// TIA Portal project "BatchSimulation_S71500_multiple_throat" (V15)

(* hardware
DEVICE "S71500/ET200MP station_1"  S7-1500 station
   slot 0: "Rail_0"  Rack  6ES7 590-1***0-0AA0
   slot 1: "PLC_2_BatchController"  CPU 1512C-1 PN  6ES7 512-1CK01-0AB0  V2.5
      slot 3: "CPU display_1"  6ES7591-1AA00-0AA0
   slot 2: "CM PtP RS422/485 HF_1"  CM PtP RS422/485 HF  6ES7 541-1AB00-0AB0  V1.0
DEVICE "S71500/ET200MP station_2"  S7-1500 station
   slot 0: "Rail_0"  Rack  6ES7 590-1***0-0AA0
   slot 1: "PLC_1_Master"  CPU 1512C-1 PN  6ES7 512-1CK01-0AB0  V2.5
      slot 3: "CPU display_1"  6ES7591-1AA00-0AA0
*)

// ===== PLC "PLC_2_BatchController"  CPU 1512C-1 PN =====

VAR_GLOBAL   // PLC tag table "Default tag table"
   "System_Byte" AT %MB1 : Byte;
   "FirstScan" AT %M1.0 : Bool;
   "DiagStatusUpdate" AT %M1.1 : Bool;
   "AlwaysTRUE" AT %M1.2 : Bool;
   "AlwaysFALSE" AT %M1.3 : Bool;
END_VAR

DATA_BLOCK "Batch1_Send"   // DB4
{ S7_Optimized_Access := 'FALSE' }
VERSION : 0.1
   VAR
      Ready : Bool;   // Batch đã sẵn sàng
      Running : Bool;   // Batch đang chạy
      Clock : Bool;   // xung trả về từ cảm biến lưu lượng
      Pulse : Int := 13;   // tổng số xung từ lúc bắt đầu chạy của cảm biến lưu lượng
      Vout : Real;   // thể tích đã xuất ra (m3)
      ctrvalue : Real;   // độ mở van (0-100%)
   END_VAR
BEGIN
END_DATA_BLOCK

DATA_BLOCK "Batch1_Recv"   // DB5
{ S7_Optimized_Access := 'FALSE' }
VERSION : 0.1
   VAR
      Start : Bool;   // tín hiệu bắt đầu chạy
      Estop : Bool;   // tín hiệu dừng khẩn cấp
      Enable : Bool;   // tín hiệu cho phép làm việc
      PS : Int;   // số xung/lit của cảm biến lưu lượng
      Setpoint : Real;   // thể tích cần xuất
   END_VAR
BEGIN
END_DATA_BLOCK

DATA_BLOCK "Batch2_Send"   // DB8
{ S7_Optimized_Access := 'FALSE' }
VERSION : 0.1
   VAR
      Ready : Bool;   // Batch đã sẵn sàng
      Running : Bool;   // Batch đang chạy
      Clock : Bool;   // xung trả về từ cảm biến lưu lượng
      Pulse : Int := 13;   // tổng số xung từ lúc bắt đầu chạy của cảm biến lưu lượng
      Vout : Real;   // thể tích đã xuất ra (m3)
      ctrvalue : Real;   // độ mở van (0-100%)
   END_VAR
BEGIN
END_DATA_BLOCK

DATA_BLOCK "Batch2_Recv"   // DB9
{ S7_Optimized_Access := 'FALSE' }
VERSION : 0.1
   VAR
      Start : Bool;   // tín hiệu bắt đầu chạy
      Estop : Bool;   // tín hiệu dừng khẩn cấp
      Enable : Bool;   // tín hiệu cho phép làm việc
      PS : Int;   // số xung/lit của cảm biến lưu lượng
      Setpoint : Real;   // thể tích cần xuất
   END_VAR
BEGIN
END_DATA_BLOCK

DATA_BLOCK "RON921_Recv"   // DB12
{ S7_Optimized_Access := 'FALSE' }
VERSION : 0.1
   VAR
      Start : Bool;   // tín hiệu bắt đầu chạy
      Estop : Bool;   // tín hiệu dừng khẩn cấp
      Enable : Bool;   // tín hiệu cho phép làm việc
      PS : Int;   // số xung/lit của cảm biến lưu lượng
      Setpoint : Real;   // thể tích cần xuất
   END_VAR
BEGIN
END_DATA_BLOCK

DATA_BLOCK "RON921_Send"   // DB13
{ S7_Optimized_Access := 'FALSE' }
VERSION : 0.1
   VAR
      Ready : Bool;   // Batch đã sẵn sàng
      Running : Bool;   // Batch đang chạy
      Clock : Bool;   // xung trả về từ cảm biến lưu lượng
      Pulse : Int := 13;   // tổng số xung từ lúc bắt đầu chạy của cảm biến lưu lượng
      Vout : Real;   // thể tích đã xuất ra (m3)
      ctrvalue : Real;   // độ mở van (0-100%)
   END_VAR
BEGIN
END_DATA_BLOCK

DATA_BLOCK "RON922_Recv"   // DB14
{ S7_Optimized_Access := 'FALSE' }
VERSION : 0.1
   VAR
      Start : Bool;   // tín hiệu bắt đầu chạy
      Estop : Bool;   // tín hiệu dừng khẩn cấp
      Enable : Bool;   // tín hiệu cho phép làm việc
      PS : Int;   // số xung/lit của cảm biến lưu lượng
      Setpoint : Real;   // thể tích cần xuất
   END_VAR
BEGIN
END_DATA_BLOCK

DATA_BLOCK "RON922_Send"   // DB15
{ S7_Optimized_Access := 'FALSE' }
VERSION : 0.1
   VAR
      Ready : Bool;   // Batch đã sẵn sàng
      Running : Bool;   // Batch đang chạy
      Clock : Bool;   // xung trả về từ cảm biến lưu lượng
      Pulse : Int := 13;   // tổng số xung từ lúc bắt đầu chạy của cảm biến lưu lượng
      Vout : Real;   // thể tích đã xuất ra (m3)
      ctrvalue : Real;   // độ mở van (0-100%)
   END_VAR
BEGIN
END_DATA_BLOCK

DATA_BLOCK "RON951_Recv"   // DB20
{ S7_Optimized_Access := 'FALSE' }
VERSION : 0.1
   VAR
      Start : Bool;   // tín hiệu bắt đầu chạy
      Estop : Bool;   // tín hiệu dừng khẩn cấp
      Enable : Bool;   // tín hiệu cho phép làm việc
      PS : Int;   // số xung/lit của cảm biến lưu lượng
      Setpoint : Real;   // thể tích cần xuất
   END_VAR
BEGIN
END_DATA_BLOCK

DATA_BLOCK "RON951_Send"   // DB21
{ S7_Optimized_Access := 'FALSE' }
VERSION : 0.1
   VAR
      Ready : Bool;   // Batch đã sẵn sàng
      Running : Bool;   // Batch đang chạy
      Clock : Bool;   // xung trả về từ cảm biến lưu lượng
      Pulse : Int := 13;   // tổng số xung từ lúc bắt đầu chạy của cảm biến lưu lượng
      Vout : Real;   // thể tích đã xuất ra (m3)
      ctrvalue : Real;   // độ mở van (0-100%)
   END_VAR
BEGIN
END_DATA_BLOCK

DATA_BLOCK "RON952_Recv"   // DB22
{ S7_Optimized_Access := 'FALSE' }
VERSION : 0.1
   VAR
      Start : Bool;   // tín hiệu bắt đầu chạy
      Estop : Bool;   // tín hiệu dừng khẩn cấp
      Enable : Bool;   // tín hiệu cho phép làm việc
      PS : Int;   // số xung/lit của cảm biến lưu lượng
      Setpoint : Real;   // thể tích cần xuất
   END_VAR
BEGIN
END_DATA_BLOCK

DATA_BLOCK "RON952_Send"   // DB23
{ S7_Optimized_Access := 'FALSE' }
VERSION : 0.1
   VAR
      Ready : Bool;   // Batch đã sẵn sàng
      Running : Bool;   // Batch đang chạy
      Clock : Bool;   // xung trả về từ cảm biến lưu lượng
      Pulse : Int := 13;   // tổng số xung từ lúc bắt đầu chạy của cảm biến lưu lượng
      Vout : Real;   // thể tích đã xuất ra (m3)
      ctrvalue : Real;   // độ mở van (0-100%)
   END_VAR
BEGIN
END_DATA_BLOCK

DATA_BLOCK "E51_Recv"   // DB28
{ S7_Optimized_Access := 'FALSE' }
VERSION : 0.1
   VAR
      Start : Bool;   // tín hiệu bắt đầu chạy
      Estop : Bool;   // tín hiệu dừng khẩn cấp
      Enable : Bool;   // tín hiệu cho phép làm việc
      PS : Int := 13;   // số xung/lit của cảm biến lưu lượng
      Setpoint : Real;   // thể tích cần xuất
   END_VAR
BEGIN
END_DATA_BLOCK

DATA_BLOCK "E51_Send"   // DB29
{ S7_Optimized_Access := 'FALSE' }
VERSION : 0.1
   VAR
      Ready : Bool;   // Batch đã sẵn sàng
      Running : Bool;   // Batch đang chạy
      ClockRON92 : Bool;   // xung trả về từ cảm biến lưu lượng
      ClockE100 : Bool;
      PulseRON92 : Int := 13;   // tổng số xung từ lúc bắt đầu chạy của cảm biến lưu lượng
      PulseE100 : Int := 13;   // tổng số xung từ lúc bắt đầu chạy của cảm biến lưu lượng
      VoutRON92 : Real;   // thể tích đã xuất ra (m3)
      VoutE100 : Real;   // thể tích đã xuất ra (m3)
      Vout : Real;   // thể tích đã xuất ra (m3)
      ctrvalueRON92 : Real;   // độ mở van (0-100%)
      ctrvalueE100 : Real;   // độ mở van (0-100%)
   END_VAR
BEGIN
END_DATA_BLOCK

DATA_BLOCK "E52_Recv"   // DB30
{ S7_Optimized_Access := 'FALSE' }
VERSION : 0.1
   VAR
      Start : Bool;   // tín hiệu bắt đầu chạy
      Estop : Bool;   // tín hiệu dừng khẩn cấp
      Enable : Bool;   // tín hiệu cho phép làm việc
      PS : Int := 13;   // số xung/lit của cảm biến lưu lượng
      Setpoint : Real;   // thể tích cần xuất
   END_VAR
BEGIN
END_DATA_BLOCK

DATA_BLOCK "E52_Send"   // DB31
{ S7_Optimized_Access := 'FALSE' }
VERSION : 0.1
   VAR
      Ready : Bool;   // Batch đã sẵn sàng
      Running : Bool;   // Batch đang chạy
      ClockRON92 : Bool;   // xung trả về từ cảm biến lưu lượng
      ClockE100 : Bool;
      PulseRON92 : Int := 13;   // tổng số xung từ lúc bắt đầu chạy của cảm biến lưu lượng
      PulseE100 : Int := 13;   // tổng số xung từ lúc bắt đầu chạy của cảm biến lưu lượng
      VoutRON92 : Real;   // thể tích đã xuất ra (m3)
      VoutE100 : Real;   // thể tích đã xuất ra (m3)
      Vout : Real;   // thể tích đã xuất ra (m3)
      ctrvalueRON92 : Real;   // độ mở van (0-100%)
      ctrvalueE100 : Real;   // độ mở van (0-100%)
   END_VAR
BEGIN
END_DATA_BLOCK

// folder: System blocks/Program resources

DATA_BLOCK "IEC_Timer_0_DB"   // DB1
{ S7_Optimized_Access := 'TRUE' }
AUTHOR : Simatic
FAMILY : IEC
NAME : IEC_TMR
VERSION : 1.0
// stored: InstanceOfName IEC_TIMER
"IEC_TIMER"
BEGIN
END_DATA_BLOCK

DATA_BLOCK "IEC_Timer_0_DB_1"   // DB2
{ S7_Optimized_Access := 'TRUE' }
AUTHOR : Simatic
FAMILY : IEC
NAME : IEC_TMR
VERSION : 1.0
// stored: InstanceOfName IEC_TIMER
"IEC_TIMER"
BEGIN
END_DATA_BLOCK

// folder: (top level)

FUNCTION "ClockGenerator" : Void   // FC1, LAD
{ S7_Optimized_Access := 'TRUE' }
VERSION : 0.1
   VAR_INPUT
      "Flow (m3/h)" : Real;
      PS : Int;
   END_VAR
   VAR_IN_OUT
      clock : Bool;
   END_VAR
   VAR_TEMP
      timing_ms : Int;
      timing : Time;
   END_VAR
BEGIN

REGION Network 1: tính ra chu kì của xung theo lưu lượng
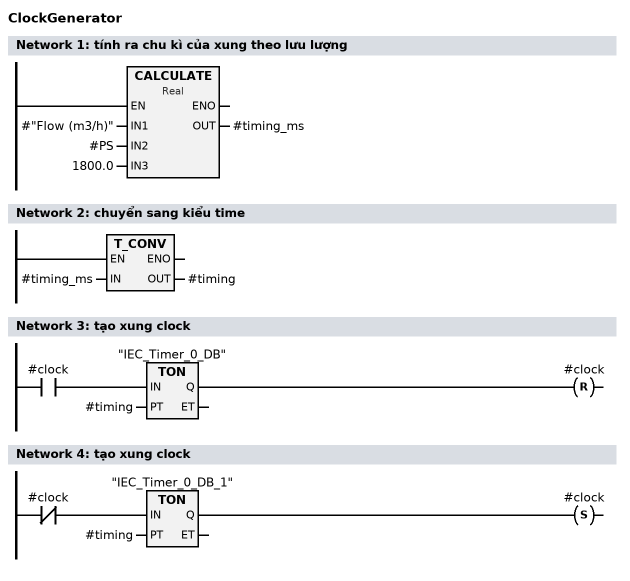
   RUNG wire#powerrail
      { S7_Templates := "SrcType := Real"; S7_Expression := "IN3/(IN1*IN2)" } Calculate(in1 := #"Flow (m3/h)", in2 := #PS, in3 := 1800.0, out => #timing_ms)
   END_RUNG
   // the same network as SCL:
   #timing_ms := 1800.0/(#"Flow (m3/h)"*#PS);
END_REGION

REGION Network 2: chuyển sang kiểu time
   #timing := T_CONV(IN := #timing_ms);
END_REGION

REGION Network 3: tạo xung clock
   "IEC_Timer_0_DB".TON(IN := #clock, PT := #timing);
   IF "IEC_Timer_0_DB".Q THEN #clock := FALSE; END_IF;
END_REGION

REGION Network 4: tạo xung clock
   "IEC_Timer_0_DB_1".TON(IN := NOT #clock, PT := #timing);
   IF "IEC_Timer_0_DB_1".Q THEN #clock := TRUE; END_IF;
END_REGION
END_FUNCTION

FUNCTION "BatchSimulation" : Void   // FC2, LAD
{ S7_Optimized_Access := 'TRUE' }
VERSION : 0.1
   VAR_INPUT
      Enable : Bool;
      Start : Bool;
      Estop : Bool;
      Setpoint : Real;
      PS : Int;
   END_VAR
   VAR_OUTPUT
      Ready : Bool;
   END_VAR
   VAR_IN_OUT
      "Vout(m3)" : Real;
      Running : Bool;
      pulse : Int;
      ctrlvalue : Real;
      clock : Bool;
   END_VAR
   VAR_TEMP
      flow : Real;
      tmp_clock : Bool;
      tmp_running : Bool;
   END_VAR
   VAR_TEMP   // added for the SCL form of the ladder/FBD networks
      _w1 : Bool;
   END_VAR
BEGIN

REGION Network 1: logic control
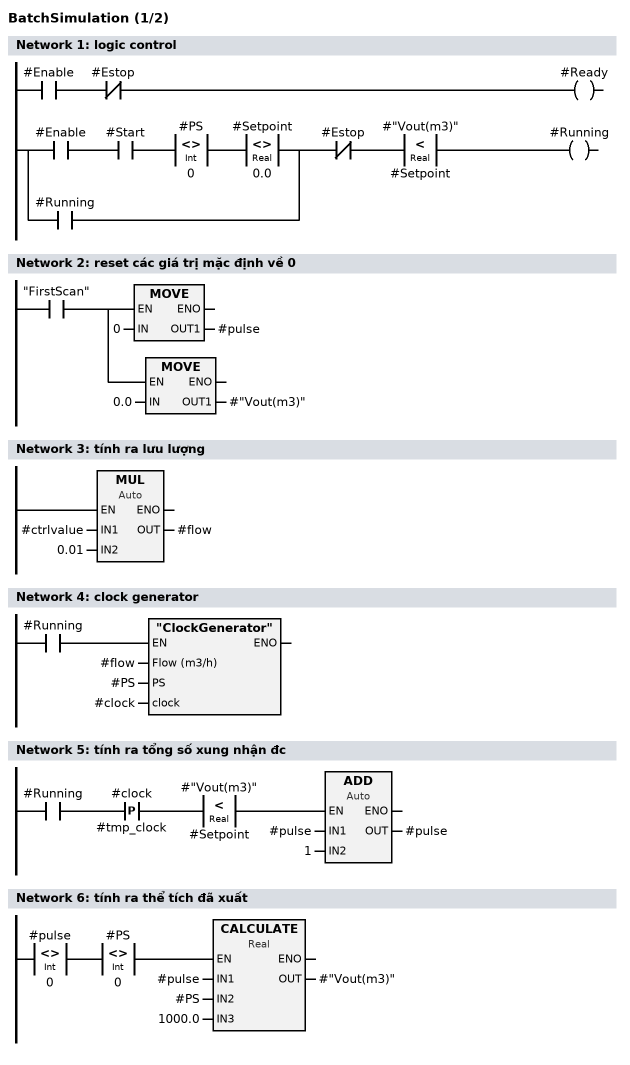
   RUNG wire#powerrail
      Contact( #Enable )
      I_Contact( #Estop )
      Coil( #Ready )
   END_RUNG
   RUNG wire#powerrail
      Contact( #Enable )
      Contact( #Start )
      { S7_Templates := "SrcType := Int" } NE_Contact(in1 := #PS, in2 := 0)
      { S7_Templates := "SrcType := Real" } NE_Contact(in1 := #Setpoint, in2 := 0.0)
      wire#w1
      I_Contact( #Estop )
      { S7_Templates := "SrcType := Real" } LT_Contact(in1 := #"Vout(m3)", in2 := #Setpoint)
      Coil( #Running )
   END_RUNG
   RUNG wire#powerrail
      Contact( #Running )
   END_RUNG wire#w1
   // the same network as SCL:
   #Ready := #Enable AND NOT #Estop;
   #Running := ((#Enable AND #Start AND (#PS <> 0) AND (#Setpoint <> 0.0)) OR #Running) AND NOT #Estop AND (#"Vout(m3)" < #Setpoint);
END_REGION

REGION Network 2: reset các giá trị mặc định về 0
   RUNG wire#powerrail
      Contact( "FirstScan" )
      wire#w1
      Move(in := 0, out1 => #pulse)
   END_RUNG
   RUNG wire#w1
      Move(in := 0.0, out1 => #"Vout(m3)")
   END_RUNG
   // the same network as SCL:
   IF "FirstScan" THEN
       #pulse := 0;
       #"Vout(m3)" := 0.0;
   END_IF;
END_REGION

REGION Network 3: tính ra lưu lượng
   RUNG wire#powerrail
      Mul(in1 := #ctrlvalue, in2 := 0.01, out => #flow)
   END_RUNG
   // the same network as SCL:
   #flow := #ctrlvalue * 0.01;
END_REGION

REGION Network 4: clock generator
   RUNG wire#powerrail
      Contact( #Running )
      "ClockGenerator"("Flow (m3/h)" := #flow, PS := #PS, clock := #clock)
   END_RUNG
   // the same network as SCL:
   IF #Running THEN "ClockGenerator"("Flow (m3/h)" := #flow, PS := #PS, clock := #clock); END_IF;
END_REGION

REGION Network 5: tính ra tổng số xung nhận đc
   RUNG wire#powerrail
      Contact( #Running )
      P_Contact(operand := #clock, bit := #tmp_clock)
      { S7_Templates := "SrcType := Real" } LT_Contact(in1 := #"Vout(m3)", in2 := #Setpoint)
      Add(in1 := #pulse, in2 := 1, out => #pulse)
   END_RUNG
   // the same network as SCL:
   #_w1 := #Running AND #clock AND NOT #tmp_clock;   // rising edge of #clock
   #tmp_clock := #clock;
   IF #_w1 AND (#"Vout(m3)" < #Setpoint) THEN #pulse := #pulse + 1; END_IF;
END_REGION

REGION Network 6: tính ra thể tích đã xuất
   RUNG wire#powerrail
      { S7_Templates := "SrcType := Int" } NE_Contact(in1 := #pulse, in2 := 0)
      { S7_Templates := "SrcType := Int" } NE_Contact(in1 := #PS, in2 := 0)
      { S7_Templates := "SrcType := Real"; S7_Expression := "(IN1/IN2)/IN3" } Calculate(in1 := #pulse, in2 := #PS, in3 := 1000.0, out => #"Vout(m3)")
   END_RUNG
   // the same network as SCL:
   IF (#pulse <> 0) AND (#PS <> 0) THEN #"Vout(m3)" := (#pulse/#PS)/1000.0; END_IF;
END_REGION

REGION Network 7: bộ PID điều khiển độ mở van
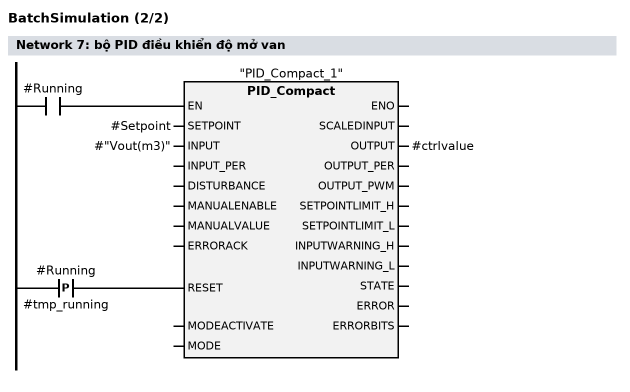
   #_w1 := #Running AND NOT #tmp_running;   // rising edge of #Running
   #tmp_running := #Running;
   IF #Running THEN
       "PID_Compact_1"(Setpoint := #Setpoint, Input := #"Vout(m3)", Reset := #_w1, Output => #ctrlvalue);   // PID_Compact
   END_IF;
END_REGION
END_FUNCTION

FUNCTION "DiezelProcess" : Void   // FC3, LAD
{ S7_Optimized_Access := 'TRUE' }
VERSION : 0.1
BEGIN

REGION Network 1: nhận dữ liệu từ DB của PLC họng 1
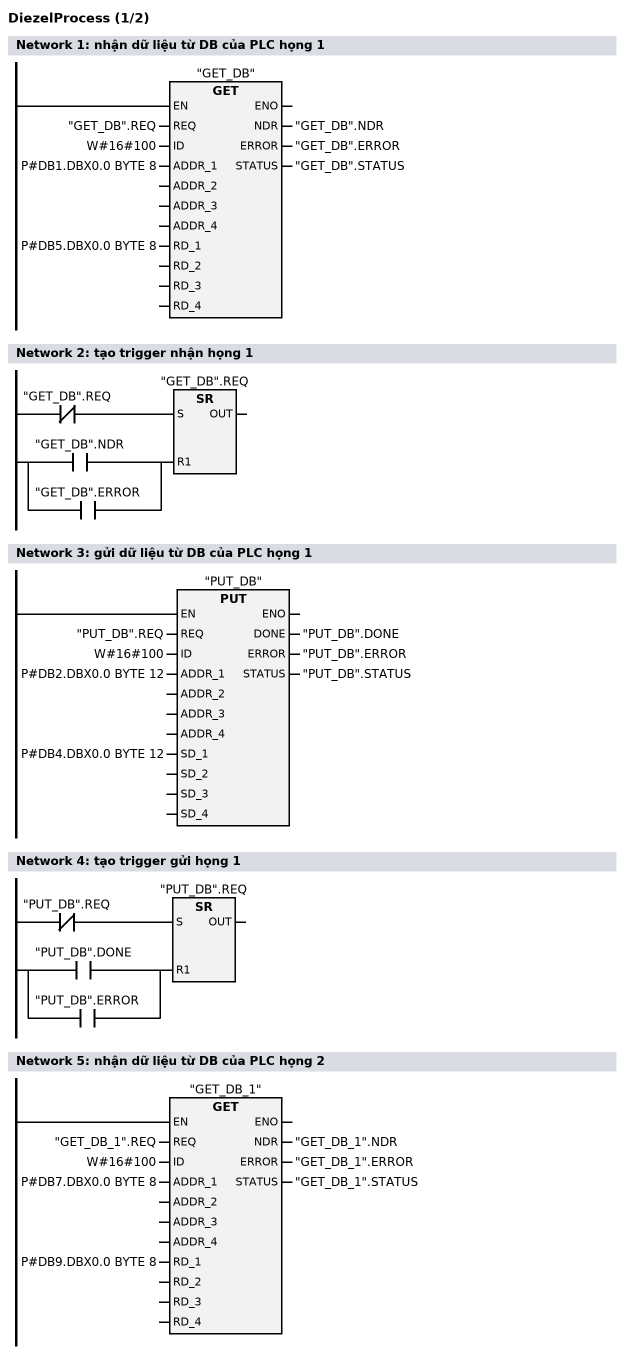
   "GET_DB"(REQ := "GET_DB".REQ,   // GET
            ID := W#16#100,
            ADDR_1 := P#DB1.DBX0.0 BYTE 8,
            RD_1 := P#DB5.DBX0.0 BYTE 8,
            NDR => "GET_DB".NDR,
            ERROR => "GET_DB".ERROR,
            STATUS => "GET_DB".STATUS);
END_REGION

REGION Network 2: tạo trigger nhận họng 1
   RUNG wire#powerrail
      I_Contact( "GET_DB".REQ )
      S_SR(operand := "GET_DB".REQ, r1 := wire#w1)
   END_RUNG
   RUNG wire#powerrail
      Contact( "GET_DB".NDR )
   END_RUNG wire#w1
   RUNG wire#powerrail
      Contact( "GET_DB".ERROR )
   END_RUNG wire#w1
   // the same network as SCL:
   IF NOT "GET_DB".REQ THEN
       "GET_DB".REQ := TRUE;   // SR flip-flop
   END_IF;
   IF "GET_DB".NDR OR "GET_DB".ERROR THEN "GET_DB".REQ := FALSE; END_IF;
END_REGION

REGION Network 3: gửi dữ liệu từ DB của PLC họng 1
   "PUT_DB"(REQ := "PUT_DB".REQ,   // PUT
            ID := W#16#100,
            ADDR_1 := P#DB2.DBX0.0 BYTE 12,
            SD_1 := P#DB4.DBX0.0 BYTE 12,
            DONE => "PUT_DB".DONE,
            ERROR => "PUT_DB".ERROR,
            STATUS => "PUT_DB".STATUS);
END_REGION

REGION Network 4: tạo trigger gửi họng 1
   RUNG wire#powerrail
      I_Contact( "PUT_DB".REQ )
      S_SR(operand := "PUT_DB".REQ, r1 := wire#w1)
   END_RUNG
   RUNG wire#powerrail
      Contact( "PUT_DB".DONE )
   END_RUNG wire#w1
   RUNG wire#powerrail
      Contact( "PUT_DB".ERROR )
   END_RUNG wire#w1
   // the same network as SCL:
   IF NOT "PUT_DB".REQ THEN
       "PUT_DB".REQ := TRUE;   // SR flip-flop
   END_IF;
   IF "PUT_DB".DONE OR "PUT_DB".ERROR THEN "PUT_DB".REQ := FALSE; END_IF;
END_REGION

REGION Network 5: nhận dữ liệu từ DB của PLC họng 2
   "GET_DB_1"(REQ := "GET_DB_1".REQ,   // GET
              ID := W#16#100,
              ADDR_1 := P#DB7.DBX0.0 BYTE 8,
              RD_1 := P#DB9.DBX0.0 BYTE 8,
              NDR => "GET_DB_1".NDR,
              ERROR => "GET_DB_1".ERROR,
              STATUS => "GET_DB_1".STATUS);
END_REGION

REGION Network 6: tạo trigger nhận họng 2
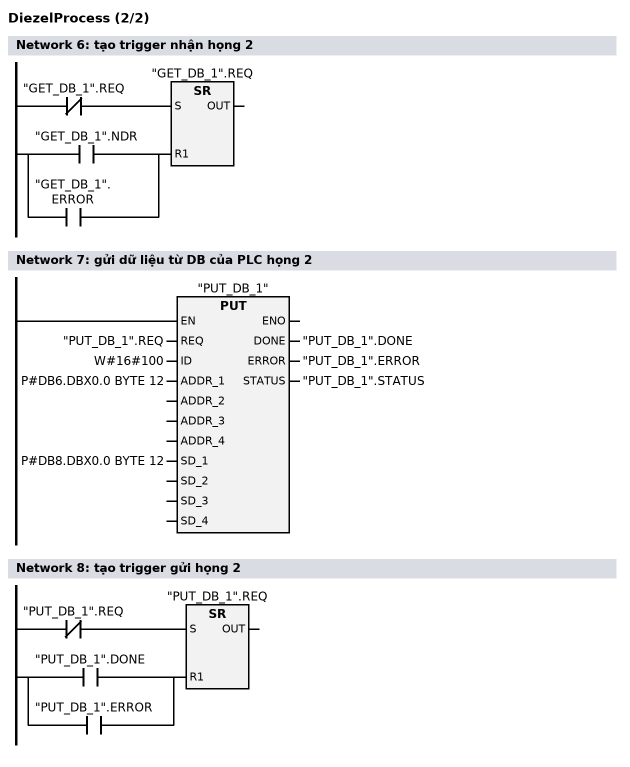
   RUNG wire#powerrail
      I_Contact( "GET_DB_1".REQ )
      S_SR(operand := "GET_DB_1".REQ, r1 := wire#w1)
   END_RUNG
   RUNG wire#powerrail
      Contact( "GET_DB_1".NDR )
   END_RUNG wire#w1
   RUNG wire#powerrail
      Contact( "GET_DB_1".ERROR )
   END_RUNG wire#w1
   // the same network as SCL:
   IF NOT "GET_DB_1".REQ THEN
       "GET_DB_1".REQ := TRUE;   // SR flip-flop
   END_IF;
   IF "GET_DB_1".NDR OR "GET_DB_1".ERROR THEN "GET_DB_1".REQ := FALSE; END_IF;
END_REGION

REGION Network 7: gửi dữ liệu từ DB của PLC họng 2
   "PUT_DB_1"(REQ := "PUT_DB_1".REQ,   // PUT
              ID := W#16#100,
              ADDR_1 := P#DB6.DBX0.0 BYTE 12,
              SD_1 := P#DB8.DBX0.0 BYTE 12,
              DONE => "PUT_DB_1".DONE,
              ERROR => "PUT_DB_1".ERROR,
              STATUS => "PUT_DB_1".STATUS);
END_REGION

REGION Network 8: tạo trigger gửi họng 2
   RUNG wire#powerrail
      I_Contact( "PUT_DB_1".REQ )
      S_SR(operand := "PUT_DB_1".REQ, r1 := wire#w1)
   END_RUNG
   RUNG wire#powerrail
      Contact( "PUT_DB_1".DONE )
   END_RUNG wire#w1
   RUNG wire#powerrail
      Contact( "PUT_DB_1".ERROR )
   END_RUNG wire#w1
   // the same network as SCL:
   IF NOT "PUT_DB_1".REQ THEN
       "PUT_DB_1".REQ := TRUE;   // SR flip-flop
   END_IF;
   IF "PUT_DB_1".DONE OR "PUT_DB_1".ERROR THEN "PUT_DB_1".REQ := FALSE; END_IF;
END_REGION
END_FUNCTION

FUNCTION "RON92Process" : Void   // FC4, LAD
{ S7_Optimized_Access := 'TRUE' }
VERSION : 0.1
BEGIN

REGION Network 1: nhận dữ liệu từ DB của PLC họng 1
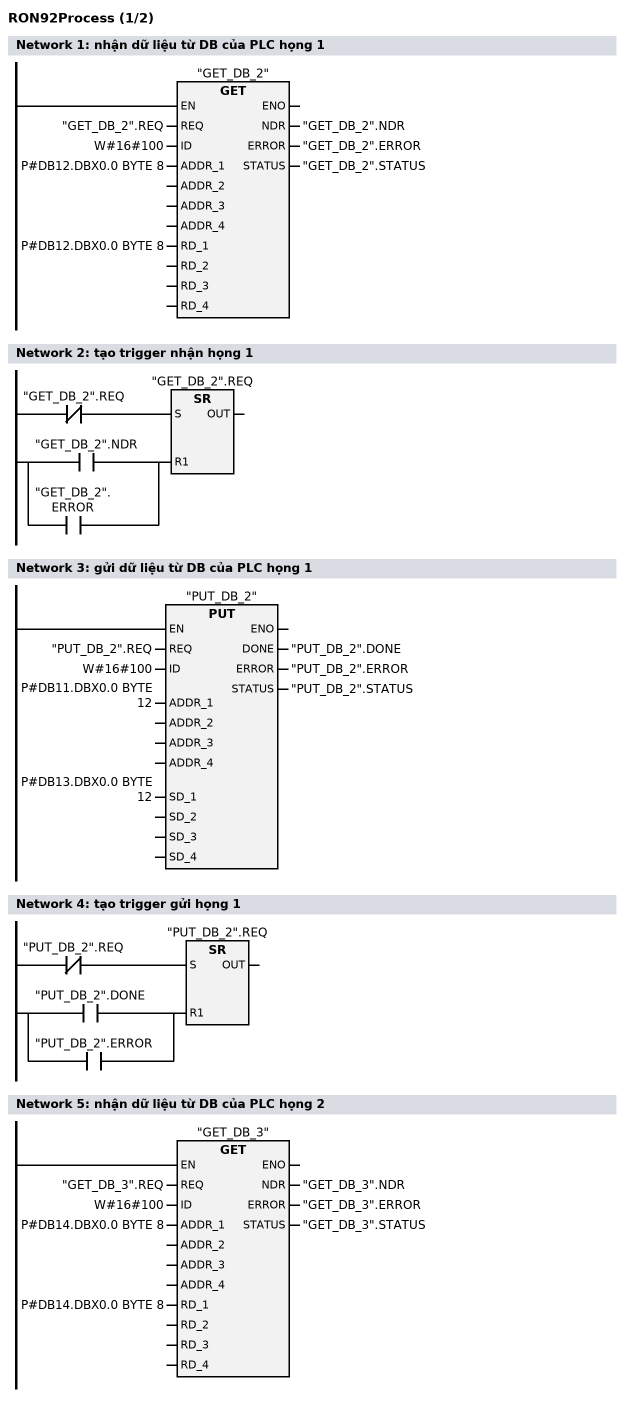
   "GET_DB_2"(REQ := "GET_DB_2".REQ,   // GET
              ID := W#16#100,
              ADDR_1 := P#DB12.DBX0.0 BYTE 8,
              RD_1 := P#DB12.DBX0.0 BYTE 8,
              NDR => "GET_DB_2".NDR,
              ERROR => "GET_DB_2".ERROR,
              STATUS => "GET_DB_2".STATUS);
END_REGION

REGION Network 2: tạo trigger nhận họng 1
   RUNG wire#powerrail
      I_Contact( "GET_DB_2".REQ )
      S_SR(operand := "GET_DB_2".REQ, r1 := wire#w1)
   END_RUNG
   RUNG wire#powerrail
      Contact( "GET_DB_2".NDR )
   END_RUNG wire#w1
   RUNG wire#powerrail
      Contact( "GET_DB_2".ERROR )
   END_RUNG wire#w1
   // the same network as SCL:
   IF NOT "GET_DB_2".REQ THEN
       "GET_DB_2".REQ := TRUE;   // SR flip-flop
   END_IF;
   IF "GET_DB_2".NDR OR "GET_DB_2".ERROR THEN "GET_DB_2".REQ := FALSE; END_IF;
END_REGION

REGION Network 3: gửi dữ liệu từ DB của PLC họng 1
   "PUT_DB_2"(REQ := "PUT_DB_2".REQ,   // PUT
              ID := W#16#100,
              ADDR_1 := P#DB11.DBX0.0 BYTE 12,
              SD_1 := P#DB13.DBX0.0 BYTE 12,
              DONE => "PUT_DB_2".DONE,
              ERROR => "PUT_DB_2".ERROR,
              STATUS => "PUT_DB_2".STATUS);
END_REGION

REGION Network 4: tạo trigger gửi họng 1
   RUNG wire#powerrail
      I_Contact( "PUT_DB_2".REQ )
      S_SR(operand := "PUT_DB_2".REQ, r1 := wire#w1)
   END_RUNG
   RUNG wire#powerrail
      Contact( "PUT_DB_2".DONE )
   END_RUNG wire#w1
   RUNG wire#powerrail
      Contact( "PUT_DB_2".ERROR )
   END_RUNG wire#w1
   // the same network as SCL:
   IF NOT "PUT_DB_2".REQ THEN
       "PUT_DB_2".REQ := TRUE;   // SR flip-flop
   END_IF;
   IF "PUT_DB_2".DONE OR "PUT_DB_2".ERROR THEN "PUT_DB_2".REQ := FALSE; END_IF;
END_REGION

REGION Network 5: nhận dữ liệu từ DB của PLC họng 2
   "GET_DB_3"(REQ := "GET_DB_3".REQ,   // GET
              ID := W#16#100,
              ADDR_1 := P#DB14.DBX0.0 BYTE 8,
              RD_1 := P#DB14.DBX0.0 BYTE 8,
              NDR => "GET_DB_3".NDR,
              ERROR => "GET_DB_3".ERROR,
              STATUS => "GET_DB_3".STATUS);
END_REGION

REGION Network 6: tạo trigger nhận họng 2
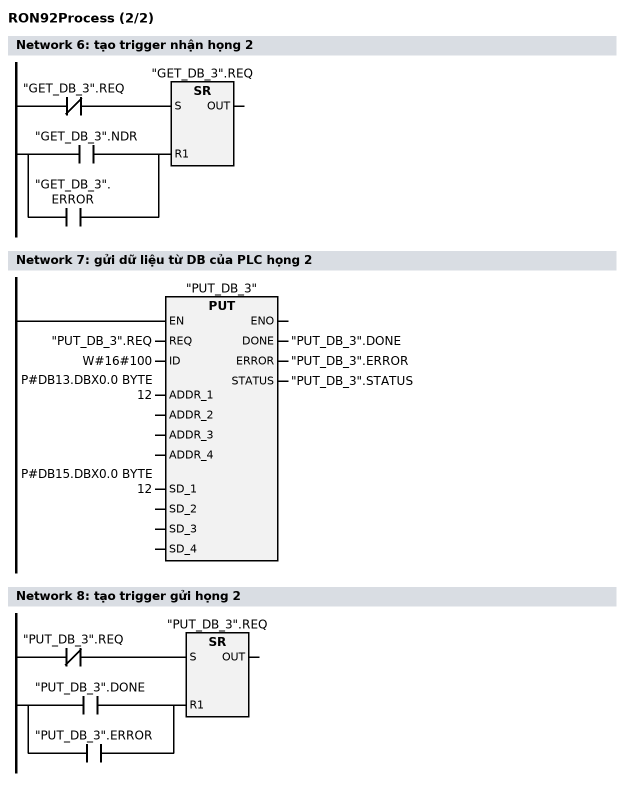
   RUNG wire#powerrail
      I_Contact( "GET_DB_3".REQ )
      S_SR(operand := "GET_DB_3".REQ, r1 := wire#w1)
   END_RUNG
   RUNG wire#powerrail
      Contact( "GET_DB_3".NDR )
   END_RUNG wire#w1
   RUNG wire#powerrail
      Contact( "GET_DB_3".ERROR )
   END_RUNG wire#w1
   // the same network as SCL:
   IF NOT "GET_DB_3".REQ THEN
       "GET_DB_3".REQ := TRUE;   // SR flip-flop
   END_IF;
   IF "GET_DB_3".NDR OR "GET_DB_3".ERROR THEN "GET_DB_3".REQ := FALSE; END_IF;
END_REGION

REGION Network 7: gửi dữ liệu từ DB của PLC họng 2
   "PUT_DB_3"(REQ := "PUT_DB_3".REQ,   // PUT
              ID := W#16#100,
              ADDR_1 := P#DB13.DBX0.0 BYTE 12,
              SD_1 := P#DB15.DBX0.0 BYTE 12,
              DONE => "PUT_DB_3".DONE,
              ERROR => "PUT_DB_3".ERROR,
              STATUS => "PUT_DB_3".STATUS);
END_REGION

REGION Network 8: tạo trigger gửi họng 2
   RUNG wire#powerrail
      I_Contact( "PUT_DB_3".REQ )
      S_SR(operand := "PUT_DB_3".REQ, r1 := wire#w1)
   END_RUNG
   RUNG wire#powerrail
      Contact( "PUT_DB_3".DONE )
   END_RUNG wire#w1
   RUNG wire#powerrail
      Contact( "PUT_DB_3".ERROR )
   END_RUNG wire#w1
   // the same network as SCL:
   IF NOT "PUT_DB_3".REQ THEN
       "PUT_DB_3".REQ := TRUE;   // SR flip-flop
   END_IF;
   IF "PUT_DB_3".DONE OR "PUT_DB_3".ERROR THEN "PUT_DB_3".REQ := FALSE; END_IF;
END_REGION
END_FUNCTION

FUNCTION "RON95Process" : Void   // FC5, LAD
{ S7_Optimized_Access := 'TRUE' }
VERSION : 0.1
BEGIN

REGION Network 1: nhận dữ liệu từ DB của PLC họng 1
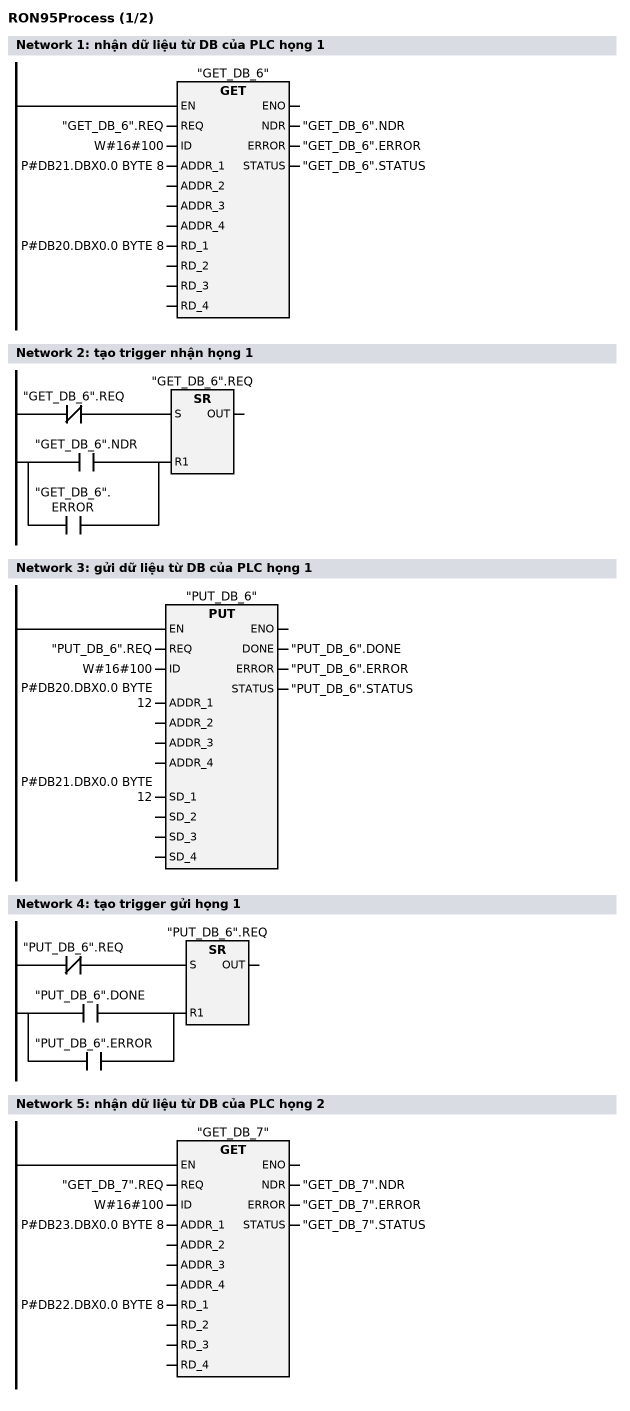
   "GET_DB_6"(REQ := "GET_DB_6".REQ,   // GET
              ID := W#16#100,
              ADDR_1 := P#DB21.DBX0.0 BYTE 8,
              RD_1 := P#DB20.DBX0.0 BYTE 8,
              NDR => "GET_DB_6".NDR,
              ERROR => "GET_DB_6".ERROR,
              STATUS => "GET_DB_6".STATUS);
END_REGION

REGION Network 2: tạo trigger nhận họng 1
   RUNG wire#powerrail
      I_Contact( "GET_DB_6".REQ )
      S_SR(operand := "GET_DB_6".REQ, r1 := wire#w1)
   END_RUNG
   RUNG wire#powerrail
      Contact( "GET_DB_6".NDR )
   END_RUNG wire#w1
   RUNG wire#powerrail
      Contact( "GET_DB_6".ERROR )
   END_RUNG wire#w1
   // the same network as SCL:
   IF NOT "GET_DB_6".REQ THEN
       "GET_DB_6".REQ := TRUE;   // SR flip-flop
   END_IF;
   IF "GET_DB_6".NDR OR "GET_DB_6".ERROR THEN "GET_DB_6".REQ := FALSE; END_IF;
END_REGION

REGION Network 3: gửi dữ liệu từ DB của PLC họng 1
   "PUT_DB_6"(REQ := "PUT_DB_6".REQ,   // PUT
              ID := W#16#100,
              ADDR_1 := P#DB20.DBX0.0 BYTE 12,
              SD_1 := P#DB21.DBX0.0 BYTE 12,
              DONE => "PUT_DB_6".DONE,
              ERROR => "PUT_DB_6".ERROR,
              STATUS => "PUT_DB_6".STATUS);
END_REGION

REGION Network 4: tạo trigger gửi họng 1
   RUNG wire#powerrail
      I_Contact( "PUT_DB_6".REQ )
      S_SR(operand := "PUT_DB_6".REQ, r1 := wire#w1)
   END_RUNG
   RUNG wire#powerrail
      Contact( "PUT_DB_6".DONE )
   END_RUNG wire#w1
   RUNG wire#powerrail
      Contact( "PUT_DB_6".ERROR )
   END_RUNG wire#w1
   // the same network as SCL:
   IF NOT "PUT_DB_6".REQ THEN
       "PUT_DB_6".REQ := TRUE;   // SR flip-flop
   END_IF;
   IF "PUT_DB_6".DONE OR "PUT_DB_6".ERROR THEN "PUT_DB_6".REQ := FALSE; END_IF;
END_REGION

REGION Network 5: nhận dữ liệu từ DB của PLC họng 2
   "GET_DB_7"(REQ := "GET_DB_7".REQ,   // GET
              ID := W#16#100,
              ADDR_1 := P#DB23.DBX0.0 BYTE 8,
              RD_1 := P#DB22.DBX0.0 BYTE 8,
              NDR => "GET_DB_7".NDR,
              ERROR => "GET_DB_7".ERROR,
              STATUS => "GET_DB_7".STATUS);
END_REGION

REGION Network 6: tạo trigger nhận họng 2
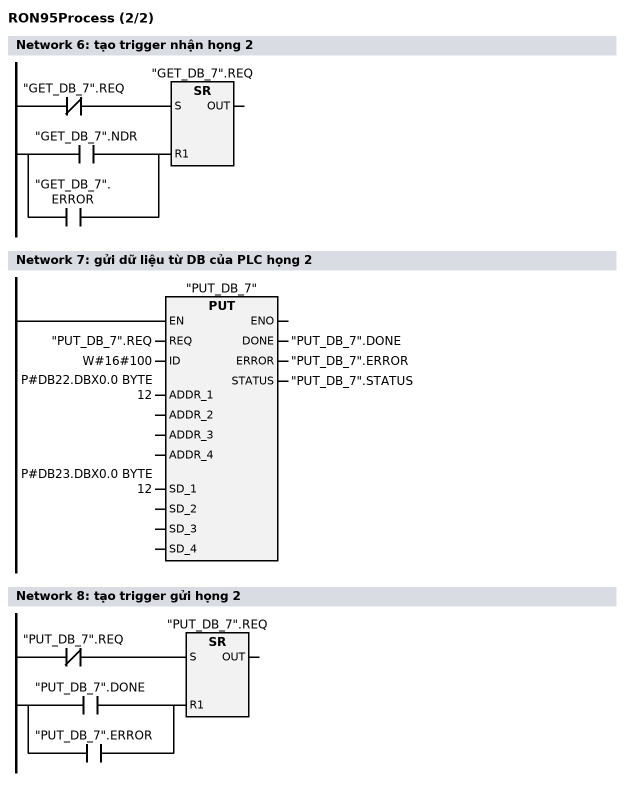
   RUNG wire#powerrail
      I_Contact( "GET_DB_7".REQ )
      S_SR(operand := "GET_DB_7".REQ, r1 := wire#w1)
   END_RUNG
   RUNG wire#powerrail
      Contact( "GET_DB_7".NDR )
   END_RUNG wire#w1
   RUNG wire#powerrail
      Contact( "GET_DB_7".ERROR )
   END_RUNG wire#w1
   // the same network as SCL:
   IF NOT "GET_DB_7".REQ THEN
       "GET_DB_7".REQ := TRUE;   // SR flip-flop
   END_IF;
   IF "GET_DB_7".NDR OR "GET_DB_7".ERROR THEN "GET_DB_7".REQ := FALSE; END_IF;
END_REGION

REGION Network 7: gửi dữ liệu từ DB của PLC họng 2
   "PUT_DB_7"(REQ := "PUT_DB_7".REQ,   // PUT
              ID := W#16#100,
              ADDR_1 := P#DB22.DBX0.0 BYTE 12,
              SD_1 := P#DB23.DBX0.0 BYTE 12,
              DONE => "PUT_DB_7".DONE,
              ERROR => "PUT_DB_7".ERROR,
              STATUS => "PUT_DB_7".STATUS);
END_REGION

REGION Network 8: tạo trigger gửi họng 2
   RUNG wire#powerrail
      I_Contact( "PUT_DB_7".REQ )
      S_SR(operand := "PUT_DB_7".REQ, r1 := wire#w1)
   END_RUNG
   RUNG wire#powerrail
      Contact( "PUT_DB_7".DONE )
   END_RUNG wire#w1
   RUNG wire#powerrail
      Contact( "PUT_DB_7".ERROR )
   END_RUNG wire#w1
   // the same network as SCL:
   IF NOT "PUT_DB_7".REQ THEN
       "PUT_DB_7".REQ := TRUE;   // SR flip-flop
   END_IF;
   IF "PUT_DB_7".DONE OR "PUT_DB_7".ERROR THEN "PUT_DB_7".REQ := FALSE; END_IF;
END_REGION
END_FUNCTION

FUNCTION "BatchSimulationE5" : Void   // FC6, LAD
{ S7_Optimized_Access := 'TRUE' }
VERSION : 0.1
   VAR_INPUT
      Enable : Bool;
      Start : Bool;
      Estop : Bool;
      Setpoint : Real;
      PS : Int;
   END_VAR
   VAR_OUTPUT
      Ready : Bool;
   END_VAR
   VAR_IN_OUT
      "Vout(m3)" : Real;
      "VoutRON92(m3)" : Real;
      "VoutE100(m3)" : Real;
      Running : Bool;
      pulseRON92 : Int;
      pulseE100 : Int;
      ctrlvalueRON92 : Real;
      ctrlvalueE100 : Real;
      clockRON92 : Bool;
      clockE100 : Bool;
   END_VAR
   VAR_TEMP
      flowRON92 : Real;
      flowE100 : Real;
      tmp_clock : Bool;
      tmp_running : Bool;
   END_VAR
   VAR_TEMP   // added for the SCL form of the ladder/FBD networks
      _w1 : Bool;
   END_VAR
BEGIN

REGION Network 1: logic control
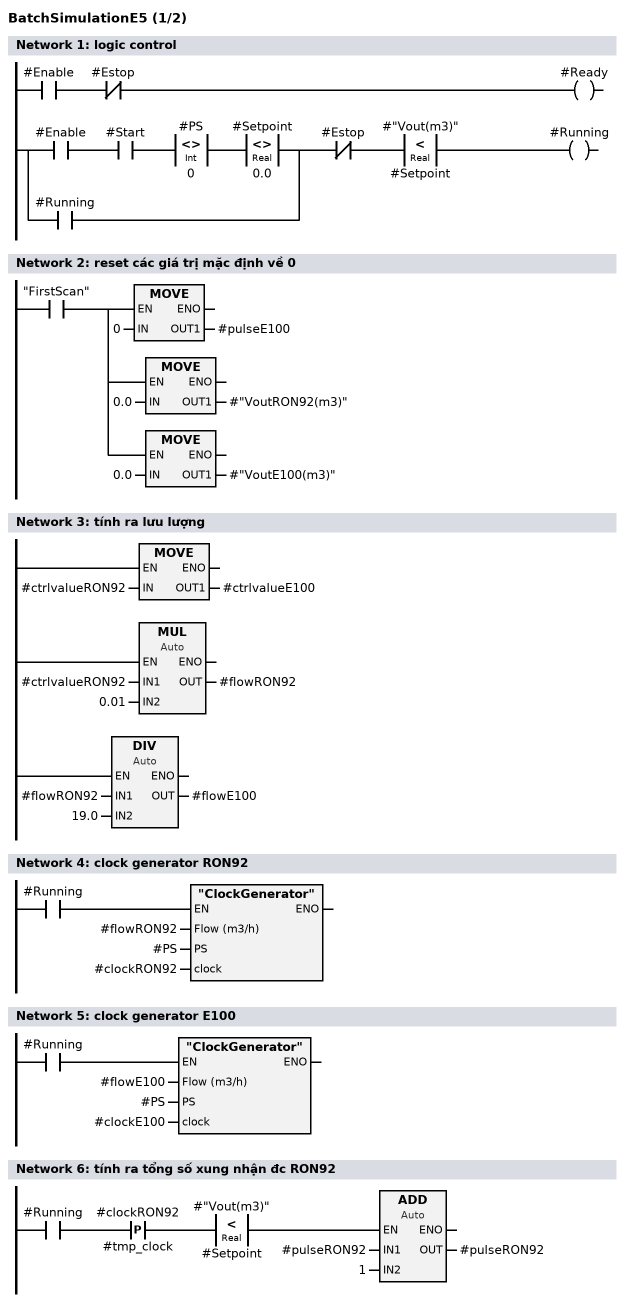
   RUNG wire#powerrail
      Contact( #Enable )
      I_Contact( #Estop )
      Coil( #Ready )
   END_RUNG
   RUNG wire#powerrail
      Contact( #Enable )
      Contact( #Start )
      { S7_Templates := "SrcType := Int" } NE_Contact(in1 := #PS, in2 := 0)
      { S7_Templates := "SrcType := Real" } NE_Contact(in1 := #Setpoint, in2 := 0.0)
      wire#w1
      I_Contact( #Estop )
      { S7_Templates := "SrcType := Real" } LT_Contact(in1 := #"Vout(m3)", in2 := #Setpoint)
      Coil( #Running )
   END_RUNG
   RUNG wire#powerrail
      Contact( #Running )
   END_RUNG wire#w1
   // the same network as SCL:
   #Ready := #Enable AND NOT #Estop;
   #Running := ((#Enable AND #Start AND (#PS <> 0) AND (#Setpoint <> 0.0)) OR #Running) AND NOT #Estop AND (#"Vout(m3)" < #Setpoint);
END_REGION

REGION Network 2: reset các giá trị mặc định về 0
   RUNG wire#powerrail
      Contact( "FirstScan" )
      wire#w1
      Move(in := 0, out1 => #pulseE100)
   END_RUNG
   RUNG wire#w1
      Move(in := 0.0, out1 => #"VoutRON92(m3)")
   END_RUNG
   RUNG wire#w1
      Move(in := 0.0, out1 => #"VoutE100(m3)")
   END_RUNG
   // the same network as SCL:
   IF "FirstScan" THEN
       #pulseE100 := 0;
       #"VoutRON92(m3)" := 0.0;
       #"VoutE100(m3)" := 0.0;
   END_IF;
END_REGION

REGION Network 3: tính ra lưu lượng
   RUNG wire#powerrail
      Move(in := #ctrlvalueRON92, out1 => #ctrlvalueE100)
   END_RUNG
   RUNG wire#powerrail
      Mul(in1 := #ctrlvalueRON92, in2 := 0.01, out => #flowRON92)
   END_RUNG
   RUNG wire#powerrail
      Div(in1 := #flowRON92, in2 := 19.0, out => #flowE100)
   END_RUNG
   // the same network as SCL:
   #ctrlvalueE100 := #ctrlvalueRON92;
   #flowRON92 := #ctrlvalueRON92 * 0.01;
   #flowE100 := #flowRON92 / 19.0;
END_REGION

REGION Network 4: clock generator RON92
   RUNG wire#powerrail
      Contact( #Running )
      "ClockGenerator"("Flow (m3/h)" := #flowRON92, PS := #PS, clock := #clockRON92)
   END_RUNG
   // the same network as SCL:
   IF #Running THEN "ClockGenerator"("Flow (m3/h)" := #flowRON92, PS := #PS, clock := #clockRON92); END_IF;
END_REGION

REGION Network 5: clock generator E100
   RUNG wire#powerrail
      Contact( #Running )
      "ClockGenerator"("Flow (m3/h)" := #flowE100, PS := #PS, clock := #clockE100)
   END_RUNG
   // the same network as SCL:
   IF #Running THEN "ClockGenerator"("Flow (m3/h)" := #flowE100, PS := #PS, clock := #clockE100); END_IF;
END_REGION

REGION Network 6: tính ra tổng số xung nhận đc RON92
   RUNG wire#powerrail
      Contact( #Running )
      P_Contact(operand := #clockRON92, bit := #tmp_clock)
      { S7_Templates := "SrcType := Real" } LT_Contact(in1 := #"Vout(m3)", in2 := #Setpoint)
      Add(in1 := #pulseRON92, in2 := 1, out => #pulseRON92)
   END_RUNG
   // the same network as SCL:
   #_w1 := #Running AND #clockRON92 AND NOT #tmp_clock;   // rising edge of #clockRON92
   #tmp_clock := #clockRON92;
   IF #_w1 AND (#"Vout(m3)" < #Setpoint) THEN #pulseRON92 := #pulseRON92 + 1; END_IF;
END_REGION

REGION Network 7: tính ra tổng số xung nhận đc E100
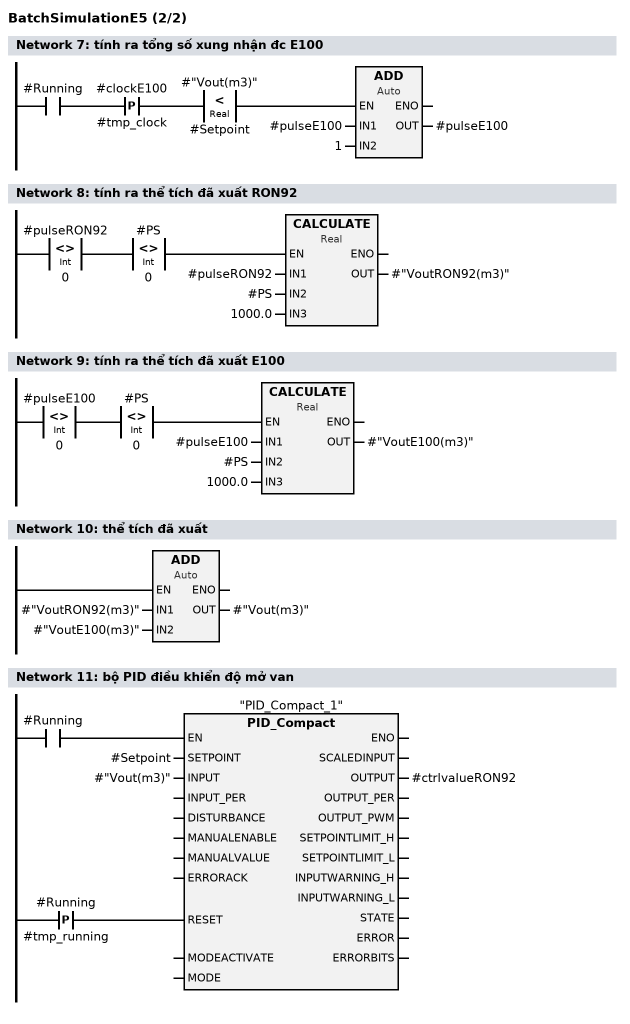
   RUNG wire#powerrail
      Contact( #Running )
      P_Contact(operand := #clockE100, bit := #tmp_clock)
      { S7_Templates := "SrcType := Real" } LT_Contact(in1 := #"Vout(m3)", in2 := #Setpoint)
      Add(in1 := #pulseE100, in2 := 1, out => #pulseE100)
   END_RUNG
   // the same network as SCL:
   #_w1 := #Running AND #clockE100 AND NOT #tmp_clock;   // rising edge of #clockE100
   #tmp_clock := #clockE100;
   IF #_w1 AND (#"Vout(m3)" < #Setpoint) THEN #pulseE100 := #pulseE100 + 1; END_IF;
END_REGION

REGION Network 8: tính ra thể tích đã xuất RON92
   RUNG wire#powerrail
      { S7_Templates := "SrcType := Int" } NE_Contact(in1 := #pulseRON92, in2 := 0)
      { S7_Templates := "SrcType := Int" } NE_Contact(in1 := #PS, in2 := 0)
      { S7_Templates := "SrcType := Real"; S7_Expression := "(IN1/IN2)/IN3" } Calculate(in1 := #pulseRON92, in2 := #PS, in3 := 1000.0, out => #"VoutRON92(m3)")
   END_RUNG
   // the same network as SCL:
   IF (#pulseRON92 <> 0) AND (#PS <> 0) THEN #"VoutRON92(m3)" := (#pulseRON92/#PS)/1000.0; END_IF;
END_REGION

REGION Network 9: tính ra thể tích đã xuất E100
   RUNG wire#powerrail
      { S7_Templates := "SrcType := Int" } NE_Contact(in1 := #pulseE100, in2 := 0)
      { S7_Templates := "SrcType := Int" } NE_Contact(in1 := #PS, in2 := 0)
      { S7_Templates := "SrcType := Real"; S7_Expression := "(IN1/IN2)/IN3" } Calculate(in1 := #pulseE100, in2 := #PS, in3 := 1000.0, out => #"VoutE100(m3)")
   END_RUNG
   // the same network as SCL:
   IF (#pulseE100 <> 0) AND (#PS <> 0) THEN #"VoutE100(m3)" := (#pulseE100/#PS)/1000.0; END_IF;
END_REGION

REGION Network 10: thể tích đã xuất
   RUNG wire#powerrail
      Add(in1 := #"VoutRON92(m3)", in2 := #"VoutE100(m3)", out => #"Vout(m3)")
   END_RUNG
   // the same network as SCL:
   #"Vout(m3)" := #"VoutRON92(m3)" + #"VoutE100(m3)";
END_REGION

REGION Network 11: bộ PID điều khiển độ mở van
   #_w1 := #Running AND NOT #tmp_running;   // rising edge of #Running
   #tmp_running := #Running;
   IF #Running THEN
       "PID_Compact_1"(Setpoint := #Setpoint, Input := #"Vout(m3)", Reset := #_w1, Output => #ctrlvalueRON92);   // PID_Compact
   END_IF;
END_REGION
END_FUNCTION

FUNCTION "E5Process" : Void   // FC7, LAD
{ S7_Optimized_Access := 'TRUE' }
VERSION : 0.1
BEGIN

REGION Network 1: nhận dữ liệu từ DB của PLC họng 1
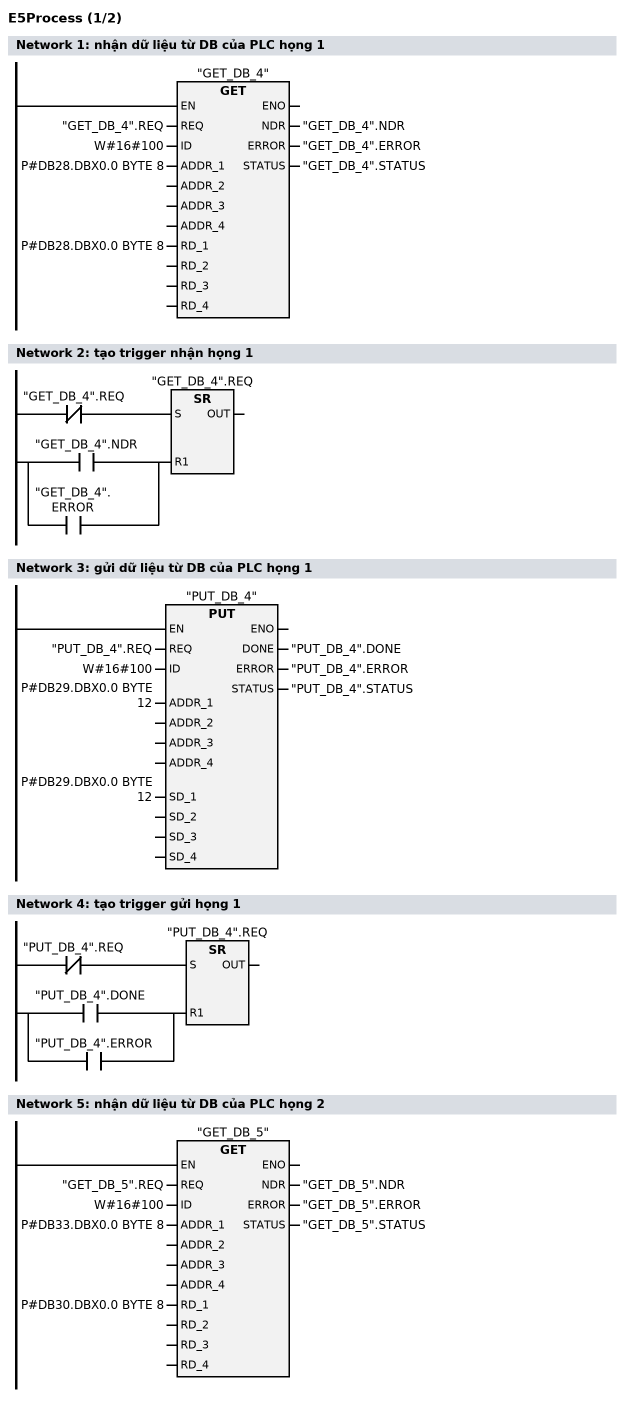
   "GET_DB_4"(REQ := "GET_DB_4".REQ,   // GET
              ID := W#16#100,
              ADDR_1 := P#DB28.DBX0.0 BYTE 8,
              RD_1 := P#DB28.DBX0.0 BYTE 8,
              NDR => "GET_DB_4".NDR,
              ERROR => "GET_DB_4".ERROR,
              STATUS => "GET_DB_4".STATUS);
END_REGION

REGION Network 2: tạo trigger nhận họng 1
   RUNG wire#powerrail
      I_Contact( "GET_DB_4".REQ )
      S_SR(operand := "GET_DB_4".REQ, r1 := wire#w1)
   END_RUNG
   RUNG wire#powerrail
      Contact( "GET_DB_4".NDR )
   END_RUNG wire#w1
   RUNG wire#powerrail
      Contact( "GET_DB_4".ERROR )
   END_RUNG wire#w1
   // the same network as SCL:
   IF NOT "GET_DB_4".REQ THEN
       "GET_DB_4".REQ := TRUE;   // SR flip-flop
   END_IF;
   IF "GET_DB_4".NDR OR "GET_DB_4".ERROR THEN "GET_DB_4".REQ := FALSE; END_IF;
END_REGION

REGION Network 3: gửi dữ liệu từ DB của PLC họng 1
   "PUT_DB_4"(REQ := "PUT_DB_4".REQ,   // PUT
              ID := W#16#100,
              ADDR_1 := P#DB29.DBX0.0 BYTE 12,
              SD_1 := P#DB29.DBX0.0 BYTE 12,
              DONE => "PUT_DB_4".DONE,
              ERROR => "PUT_DB_4".ERROR,
              STATUS => "PUT_DB_4".STATUS);
END_REGION

REGION Network 4: tạo trigger gửi họng 1
   RUNG wire#powerrail
      I_Contact( "PUT_DB_4".REQ )
      S_SR(operand := "PUT_DB_4".REQ, r1 := wire#w1)
   END_RUNG
   RUNG wire#powerrail
      Contact( "PUT_DB_4".DONE )
   END_RUNG wire#w1
   RUNG wire#powerrail
      Contact( "PUT_DB_4".ERROR )
   END_RUNG wire#w1
   // the same network as SCL:
   IF NOT "PUT_DB_4".REQ THEN
       "PUT_DB_4".REQ := TRUE;   // SR flip-flop
   END_IF;
   IF "PUT_DB_4".DONE OR "PUT_DB_4".ERROR THEN "PUT_DB_4".REQ := FALSE; END_IF;
END_REGION

REGION Network 5: nhận dữ liệu từ DB của PLC họng 2
   "GET_DB_5"(REQ := "GET_DB_5".REQ,   // GET
              ID := W#16#100,
              ADDR_1 := P#DB33.DBX0.0 BYTE 8,
              RD_1 := P#DB30.DBX0.0 BYTE 8,
              NDR => "GET_DB_5".NDR,
              ERROR => "GET_DB_5".ERROR,
              STATUS => "GET_DB_5".STATUS);
END_REGION

REGION Network 6: tạo trigger nhận họng 2
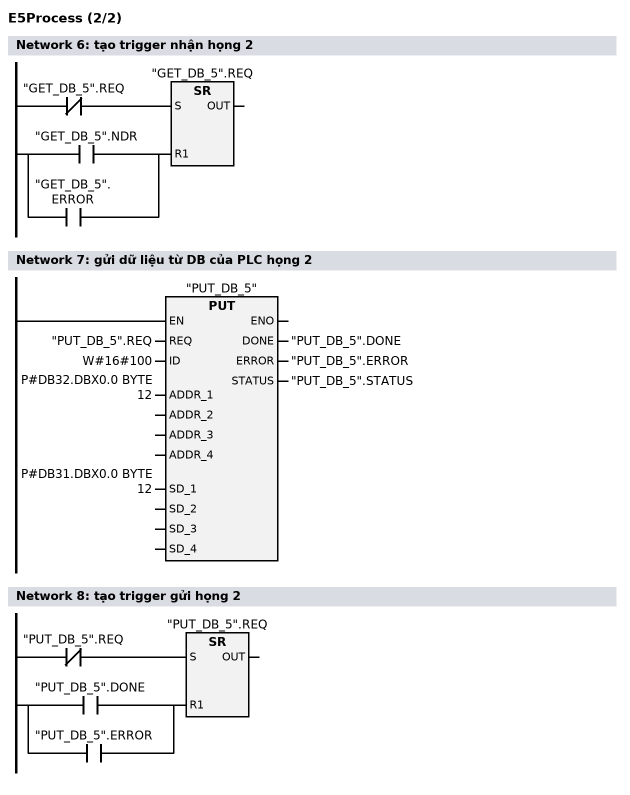
   RUNG wire#powerrail
      I_Contact( "GET_DB_5".REQ )
      S_SR(operand := "GET_DB_5".REQ, r1 := wire#w1)
   END_RUNG
   RUNG wire#powerrail
      Contact( "GET_DB_5".NDR )
   END_RUNG wire#w1
   RUNG wire#powerrail
      Contact( "GET_DB_5".ERROR )
   END_RUNG wire#w1
   // the same network as SCL:
   IF NOT "GET_DB_5".REQ THEN
       "GET_DB_5".REQ := TRUE;   // SR flip-flop
   END_IF;
   IF "GET_DB_5".NDR OR "GET_DB_5".ERROR THEN "GET_DB_5".REQ := FALSE; END_IF;
END_REGION

REGION Network 7: gửi dữ liệu từ DB của PLC họng 2
   "PUT_DB_5"(REQ := "PUT_DB_5".REQ,   // PUT
              ID := W#16#100,
              ADDR_1 := P#DB32.DBX0.0 BYTE 12,
              SD_1 := P#DB31.DBX0.0 BYTE 12,
              DONE => "PUT_DB_5".DONE,
              ERROR => "PUT_DB_5".ERROR,
              STATUS => "PUT_DB_5".STATUS);
END_REGION

REGION Network 8: tạo trigger gửi họng 2
   RUNG wire#powerrail
      I_Contact( "PUT_DB_5".REQ )
      S_SR(operand := "PUT_DB_5".REQ, r1 := wire#w1)
   END_RUNG
   RUNG wire#powerrail
      Contact( "PUT_DB_5".DONE )
   END_RUNG wire#w1
   RUNG wire#powerrail
      Contact( "PUT_DB_5".ERROR )
   END_RUNG wire#w1
   // the same network as SCL:
   IF NOT "PUT_DB_5".REQ THEN
       "PUT_DB_5".REQ := TRUE;   // SR flip-flop
   END_IF;
   IF "PUT_DB_5".DONE OR "PUT_DB_5".ERROR THEN "PUT_DB_5".REQ := FALSE; END_IF;
END_REGION
END_FUNCTION

ORGANIZATION_BLOCK "Main"   // OB1, LAD, ProgramCycle
TITLE = "Main Program Sweep (Cycle)"
{ S7_Optimized_Access := 'TRUE' }
VERSION : 0.1
   VAR_INPUT
      Initial_Call : Bool;   // Initial call of this OB
      Remanence : Bool;   // =True, if remanent data are available
   END_VAR
BEGIN

REGION Network 1: chương trình xử lý bể Diezel
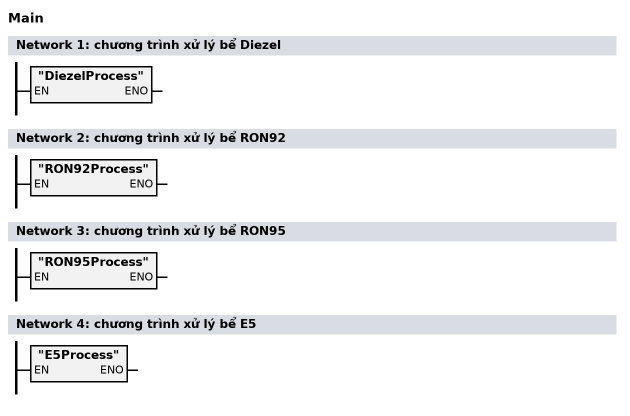
   RUNG wire#powerrail
      "DiezelProcess"()
   END_RUNG
   // the same network as SCL:
   "DiezelProcess"();
END_REGION

REGION Network 2: chương trình xử lý bể RON92
   RUNG wire#powerrail
      "RON92Process"()
   END_RUNG
   // the same network as SCL:
   "RON92Process"();
END_REGION

REGION Network 3: chương trình xử lý bể RON95
   RUNG wire#powerrail
      "RON95Process"()
   END_RUNG
   // the same network as SCL:
   "RON95Process"();
END_REGION

REGION Network 4: chương trình xử lý bể E5
   RUNG wire#powerrail
      "E5Process"()
   END_RUNG
   // the same network as SCL:
   "E5Process"();
END_REGION
END_ORGANIZATION_BLOCK

ORGANIZATION_BLOCK "Cyclic interrupt"   // OB30, LAD, CyclicInterrupt
{ S7_Optimized_Access := 'TRUE' }
VERSION : 0.1
   VAR_INPUT
      Initial_Call : Bool;   // Initial call of this OB
      Event_Count : Int;   // Events discarded
   END_VAR
BEGIN

REGION Network 1: chương trình BatchController Diezel họng 1
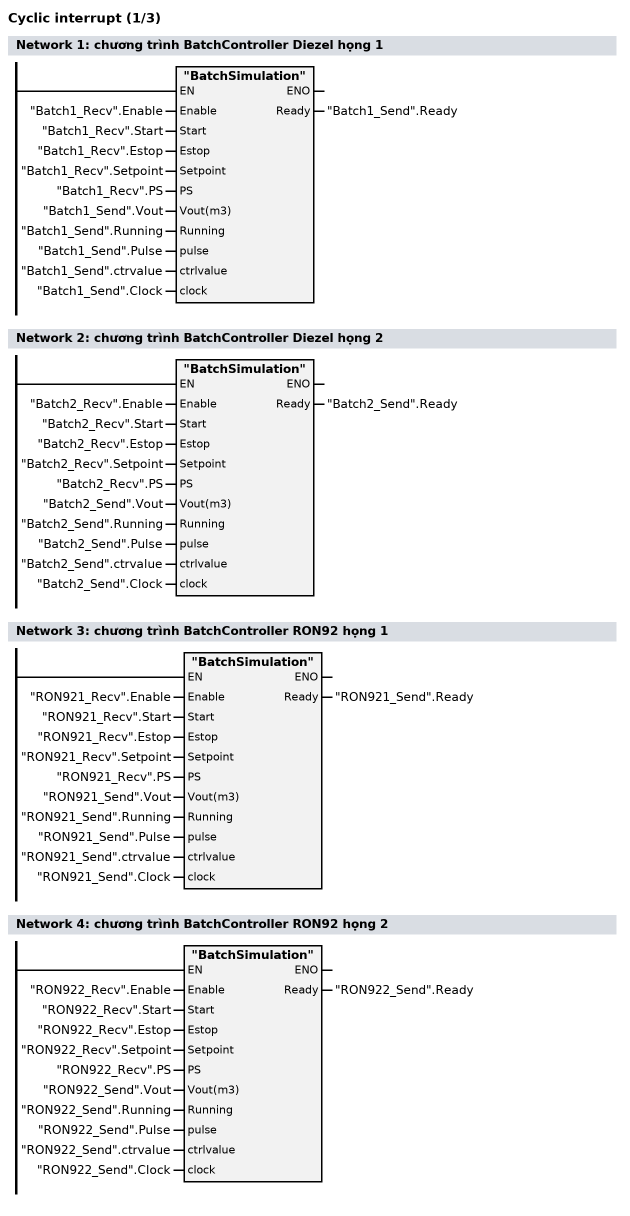
   RUNG wire#powerrail
      "BatchSimulation"(Enable := "Batch1_Recv".Enable, Start := "Batch1_Recv".Start, Estop := "Batch1_Recv".Estop, Setpoint := "Batch1_Recv".Setpoint, PS := "Batch1_Recv".PS, "Vout(m3)" := "Batch1_Send".Vout, Running := "Batch1_Send".Running, pulse := "Batch1_Send".Pulse, ctrlvalue := "Batch1_Send".ctrvalue, clock := "Batch1_Send".Clock, Ready => "Batch1_Send".Ready)
   END_RUNG
   // the same network as SCL:
   "BatchSimulation"(Enable := "Batch1_Recv".Enable,
                     Start := "Batch1_Recv".Start,
                     Estop := "Batch1_Recv".Estop,
                     Setpoint := "Batch1_Recv".Setpoint,
                     PS := "Batch1_Recv".PS,
                     "Vout(m3)" := "Batch1_Send".Vout,
                     Running := "Batch1_Send".Running,
                     pulse := "Batch1_Send".Pulse,
                     ctrlvalue := "Batch1_Send".ctrvalue,
                     clock := "Batch1_Send".Clock,
                     Ready => "Batch1_Send".Ready);
END_REGION

REGION Network 2: chương trình BatchController Diezel họng 2
   RUNG wire#powerrail
      "BatchSimulation"(Enable := "Batch2_Recv".Enable, Start := "Batch2_Recv".Start, Estop := "Batch2_Recv".Estop, Setpoint := "Batch2_Recv".Setpoint, PS := "Batch2_Recv".PS, "Vout(m3)" := "Batch2_Send".Vout, Running := "Batch2_Send".Running, pulse := "Batch2_Send".Pulse, ctrlvalue := "Batch2_Send".ctrvalue, clock := "Batch2_Send".Clock, Ready => "Batch2_Send".Ready)
   END_RUNG
   // the same network as SCL:
   "BatchSimulation"(Enable := "Batch2_Recv".Enable,
                     Start := "Batch2_Recv".Start,
                     Estop := "Batch2_Recv".Estop,
                     Setpoint := "Batch2_Recv".Setpoint,
                     PS := "Batch2_Recv".PS,
                     "Vout(m3)" := "Batch2_Send".Vout,
                     Running := "Batch2_Send".Running,
                     pulse := "Batch2_Send".Pulse,
                     ctrlvalue := "Batch2_Send".ctrvalue,
                     clock := "Batch2_Send".Clock,
                     Ready => "Batch2_Send".Ready);
END_REGION

REGION Network 3: chương trình BatchController RON92 họng 1
   RUNG wire#powerrail
      "BatchSimulation"(Enable := "RON921_Recv".Enable, Start := "RON921_Recv".Start, Estop := "RON921_Recv".Estop, Setpoint := "RON921_Recv".Setpoint, PS := "RON921_Recv".PS, "Vout(m3)" := "RON921_Send".Vout, Running := "RON921_Send".Running, pulse := "RON921_Send".Pulse, ctrlvalue := "RON921_Send".ctrvalue, clock := "RON921_Send".Clock, Ready => "RON921_Send".Ready)
   END_RUNG
   // the same network as SCL:
   "BatchSimulation"(Enable := "RON921_Recv".Enable,
                     Start := "RON921_Recv".Start,
                     Estop := "RON921_Recv".Estop,
                     Setpoint := "RON921_Recv".Setpoint,
                     PS := "RON921_Recv".PS,
                     "Vout(m3)" := "RON921_Send".Vout,
                     Running := "RON921_Send".Running,
                     pulse := "RON921_Send".Pulse,
                     ctrlvalue := "RON921_Send".ctrvalue,
                     clock := "RON921_Send".Clock,
                     Ready => "RON921_Send".Ready);
END_REGION

REGION Network 4: chương trình BatchController RON92 họng 2
   RUNG wire#powerrail
      "BatchSimulation"(Enable := "RON922_Recv".Enable, Start := "RON922_Recv".Start, Estop := "RON922_Recv".Estop, Setpoint := "RON922_Recv".Setpoint, PS := "RON922_Recv".PS, "Vout(m3)" := "RON922_Send".Vout, Running := "RON922_Send".Running, pulse := "RON922_Send".Pulse, ctrlvalue := "RON922_Send".ctrvalue, clock := "RON922_Send".Clock, Ready => "RON922_Send".Ready)
   END_RUNG
   // the same network as SCL:
   "BatchSimulation"(Enable := "RON922_Recv".Enable,
                     Start := "RON922_Recv".Start,
                     Estop := "RON922_Recv".Estop,
                     Setpoint := "RON922_Recv".Setpoint,
                     PS := "RON922_Recv".PS,
                     "Vout(m3)" := "RON922_Send".Vout,
                     Running := "RON922_Send".Running,
                     pulse := "RON922_Send".Pulse,
                     ctrlvalue := "RON922_Send".ctrvalue,
                     clock := "RON922_Send".Clock,
                     Ready => "RON922_Send".Ready);
END_REGION

REGION Network 5: chương trình BatchController RON95 họng 1
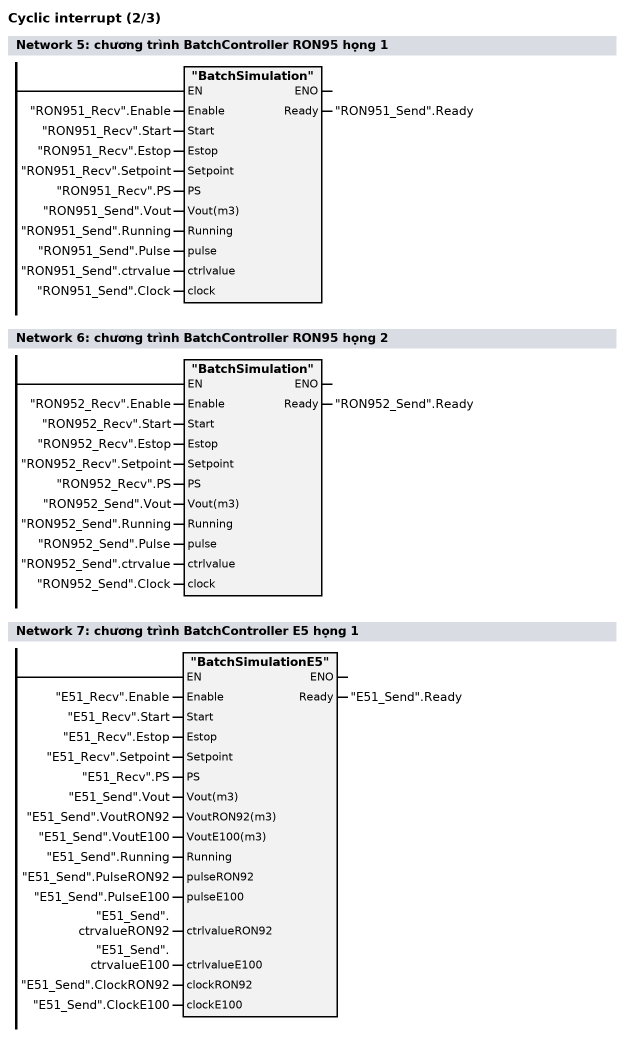
   RUNG wire#powerrail
      "BatchSimulation"(Enable := "RON951_Recv".Enable, Start := "RON951_Recv".Start, Estop := "RON951_Recv".Estop, Setpoint := "RON951_Recv".Setpoint, PS := "RON951_Recv".PS, "Vout(m3)" := "RON951_Send".Vout, Running := "RON951_Send".Running, pulse := "RON951_Send".Pulse, ctrlvalue := "RON951_Send".ctrvalue, clock := "RON951_Send".Clock, Ready => "RON951_Send".Ready)
   END_RUNG
   // the same network as SCL:
   "BatchSimulation"(Enable := "RON951_Recv".Enable,
                     Start := "RON951_Recv".Start,
                     Estop := "RON951_Recv".Estop,
                     Setpoint := "RON951_Recv".Setpoint,
                     PS := "RON951_Recv".PS,
                     "Vout(m3)" := "RON951_Send".Vout,
                     Running := "RON951_Send".Running,
                     pulse := "RON951_Send".Pulse,
                     ctrlvalue := "RON951_Send".ctrvalue,
                     clock := "RON951_Send".Clock,
                     Ready => "RON951_Send".Ready);
END_REGION

REGION Network 6: chương trình BatchController RON95 họng 2
   RUNG wire#powerrail
      "BatchSimulation"(Enable := "RON952_Recv".Enable, Start := "RON952_Recv".Start, Estop := "RON952_Recv".Estop, Setpoint := "RON952_Recv".Setpoint, PS := "RON952_Recv".PS, "Vout(m3)" := "RON952_Send".Vout, Running := "RON952_Send".Running, pulse := "RON952_Send".Pulse, ctrlvalue := "RON952_Send".ctrvalue, clock := "RON952_Send".Clock, Ready => "RON952_Send".Ready)
   END_RUNG
   // the same network as SCL:
   "BatchSimulation"(Enable := "RON952_Recv".Enable,
                     Start := "RON952_Recv".Start,
                     Estop := "RON952_Recv".Estop,
                     Setpoint := "RON952_Recv".Setpoint,
                     PS := "RON952_Recv".PS,
                     "Vout(m3)" := "RON952_Send".Vout,
                     Running := "RON952_Send".Running,
                     pulse := "RON952_Send".Pulse,
                     ctrlvalue := "RON952_Send".ctrvalue,
                     clock := "RON952_Send".Clock,
                     Ready => "RON952_Send".Ready);
END_REGION

REGION Network 7: chương trình BatchController E5 họng 1
   RUNG wire#powerrail
      "BatchSimulationE5"(Enable := "E51_Recv".Enable, Start := "E51_Recv".Start, Estop := "E51_Recv".Estop, Setpoint := "E51_Recv".Setpoint, PS := "E51_Recv".PS, "Vout(m3)" := "E51_Send".Vout, "VoutRON92(m3)" := "E51_Send".VoutRON92, "VoutE100(m3)" := "E51_Send".VoutE100, Running := "E51_Send".Running, pulseRON92 := "E51_Send".PulseRON92, pulseE100 := "E51_Send".PulseE100, ctrlvalueRON92 := "E51_Send".ctrvalueRON92, ctrlvalueE100 := "E51_Send".ctrvalueE100, clockRON92 := "E51_Send".ClockRON92, clockE100 := "E51_Send".ClockE100, Ready => "E51_Send".Ready)
   END_RUNG
   // the same network as SCL:
   "BatchSimulationE5"(Enable := "E51_Recv".Enable,
                       Start := "E51_Recv".Start,
                       Estop := "E51_Recv".Estop,
                       Setpoint := "E51_Recv".Setpoint,
                       PS := "E51_Recv".PS,
                       "Vout(m3)" := "E51_Send".Vout,
                       "VoutRON92(m3)" := "E51_Send".VoutRON92,
                       "VoutE100(m3)" := "E51_Send".VoutE100,
                       Running := "E51_Send".Running,
                       pulseRON92 := "E51_Send".PulseRON92,
                       pulseE100 := "E51_Send".PulseE100,
                       ctrlvalueRON92 := "E51_Send".ctrvalueRON92,
                       ctrlvalueE100 := "E51_Send".ctrvalueE100,
                       clockRON92 := "E51_Send".ClockRON92,
                       clockE100 := "E51_Send".ClockE100,
                       Ready => "E51_Send".Ready);
END_REGION

REGION Network 8: chương trình BatchController E5 họng 2
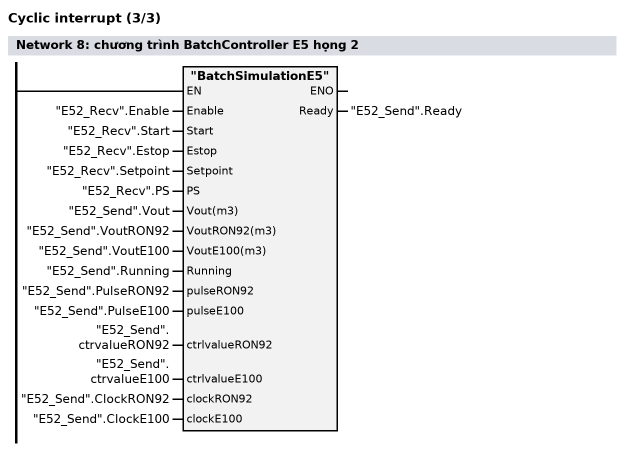
   RUNG wire#powerrail
      "BatchSimulationE5"(Enable := "E52_Recv".Enable, Start := "E52_Recv".Start, Estop := "E52_Recv".Estop, Setpoint := "E52_Recv".Setpoint, PS := "E52_Recv".PS, "Vout(m3)" := "E52_Send".Vout, "VoutRON92(m3)" := "E52_Send".VoutRON92, "VoutE100(m3)" := "E52_Send".VoutE100, Running := "E52_Send".Running, pulseRON92 := "E52_Send".PulseRON92, pulseE100 := "E52_Send".PulseE100, ctrlvalueRON92 := "E52_Send".ctrvalueRON92, ctrlvalueE100 := "E52_Send".ctrvalueE100, clockRON92 := "E52_Send".ClockRON92, clockE100 := "E52_Send".ClockE100, Ready => "E52_Send".Ready)
   END_RUNG
   // the same network as SCL:
   "BatchSimulationE5"(Enable := "E52_Recv".Enable,
                       Start := "E52_Recv".Start,
                       Estop := "E52_Recv".Estop,
                       Setpoint := "E52_Recv".Setpoint,
                       PS := "E52_Recv".PS,
                       "Vout(m3)" := "E52_Send".Vout,
                       "VoutRON92(m3)" := "E52_Send".VoutRON92,
                       "VoutE100(m3)" := "E52_Send".VoutE100,
                       Running := "E52_Send".Running,
                       pulseRON92 := "E52_Send".PulseRON92,
                       pulseE100 := "E52_Send".PulseE100,
                       ctrlvalueRON92 := "E52_Send".ctrvalueRON92,
                       ctrlvalueE100 := "E52_Send".ctrvalueE100,
                       clockRON92 := "E52_Send".ClockRON92,
                       clockE100 := "E52_Send".ClockE100,
                       Ready => "E52_Send".Ready);
END_REGION
END_ORGANIZATION_BLOCK

// ===== PLC "PLC_1_Master"  CPU 1512C-1 PN =====

DATA_BLOCK "Diezel1_Send"   // DB1
{ S7_Optimized_Access := 'FALSE' }
VERSION : 0.1
   VAR
      Start : Bool;   // tín hiệu bắt đầu chạy
      Estop : Bool;   // tín hiệu dừng khẩn cấp
      Enable : Bool;   // tín hiệu cho phép làm việc
      PS : Int := 13;   // số xung/lit của cảm biến lưu lượng
      Setpoint : Real;   // thể tích cần xuất
   END_VAR
BEGIN
END_DATA_BLOCK

DATA_BLOCK "Diezel1_Recv"   // DB2
{ S7_Optimized_Access := 'FALSE' }
VERSION : 0.1
   VAR
      Ready : Bool;   // Batch đã sẵn sàng
      Running : Bool;   // Batch đang chạy
      Clock : Bool;   // xung trả về từ cảm biến lưu lượng
      Pulse : Int := 13;   // tổng số xung từ lúc bắt đầu chạy của cảm biến lưu lượng
      Vout : Real;   // thể tích đã xuất ra (m3)
      ctrvalue : Real;   // độ mở van (0-100%)
   END_VAR
BEGIN
END_DATA_BLOCK

DATA_BLOCK "Diezel_Common"   // DB5
{ S7_Optimized_Access := 'FALSE' }
VERSION : 0.1
   VAR
      Temp : Real := 25.0;   // nhiệt độ (°C)
      Level : Real := 15.0;   // mức (m)
      InitialLevel : Real := 15.0;   // mức ban đầu (m)
      BaseArea : Real := 10.0;   // diện tích đáy (m2)
      Volume : Real;   // thể tích hiện tại (m3)
      InitialVolume : Real;   // thể tích ban đầu (m3)
      Flow1 : Real := 0.0;   // lưu lượng họng 1 (m3/h)
      Flow2 : Real := 0.0;   // lưu lượng họng 2 (m3/h)
   END_VAR
BEGIN
END_DATA_BLOCK

DATA_BLOCK "Diezel2_Recv"   // DB6
{ S7_Optimized_Access := 'FALSE' }
VERSION : 0.1
   VAR
      Ready : Bool;   // Batch đã sẵn sàng
      Running : Bool;   // Batch đang chạy
      Clock : Bool;   // xung trả về từ cảm biến lưu lượng
      Pulse : Int := 13;   // tổng số xung từ lúc bắt đầu chạy của cảm biến lưu lượng
      Vout : Real;   // thể tích đã xuất ra (m3)
      ctrvalue : Real;   // độ mở van (0-100%)
   END_VAR
BEGIN
END_DATA_BLOCK

DATA_BLOCK "Diezel2_Send"   // DB7
{ S7_Optimized_Access := 'FALSE' }
VERSION : 0.1
   VAR
      Start : Bool;   // tín hiệu bắt đầu chạy
      Estop : Bool;   // tín hiệu dừng khẩn cấp
      Enable : Bool;   // tín hiệu cho phép làm việc
      PS : Int := 13;   // số xung/lit của cảm biến lưu lượng
      Setpoint : Real;   // thể tích cần xuất
   END_VAR
BEGIN
END_DATA_BLOCK

DATA_BLOCK "RON92_Common"   // DB10
{ S7_Optimized_Access := 'FALSE' }
VERSION : 0.1
   VAR
      Temp : Real := 25.0;   // nhiệt độ (°C)
      Level : Real := 15.0;   // mức (m)
      InitialLevel : Real := 15.0;   // mức ban đầu (m)
      BaseArea : Real := 10.0;   // diện tích đáy (m2)
      Volume : Real;   // thể tích hiện tại (m3)
      InitialVolume : Real;   // thể tích ban đầu (m3)
      Flow1 : Real := 0.0;   // lưu lượng họng 1 (m3/h)
      Flow2 : Real := 0.0;   // lưu lượng họng 2 (m3/h)
   END_VAR
BEGIN
END_DATA_BLOCK

DATA_BLOCK "RON921_Recv"   // DB11
{ S7_Optimized_Access := 'FALSE' }
VERSION : 0.1
   VAR
      Ready : Bool;   // Batch đã sẵn sàng
      Running : Bool;   // Batch đang chạy
      Clock : Bool;   // xung trả về từ cảm biến lưu lượng
      Pulse : Int := 13;   // tổng số xung từ lúc bắt đầu chạy của cảm biến lưu lượng
      Vout : Real;   // thể tích đã xuất ra (m3)
      ctrvalue : Real;   // độ mở van (0-100%)
   END_VAR
BEGIN
END_DATA_BLOCK

DATA_BLOCK "RON921_Send"   // DB12
{ S7_Optimized_Access := 'FALSE' }
VERSION : 0.1
   VAR
      Start : Bool;   // tín hiệu bắt đầu chạy
      Estop : Bool;   // tín hiệu dừng khẩn cấp
      Enable : Bool;   // tín hiệu cho phép làm việc
      PS : Int := 13;   // số xung/lit của cảm biến lưu lượng
      Setpoint : Real;   // thể tích cần xuất
   END_VAR
BEGIN
END_DATA_BLOCK

DATA_BLOCK "RON922_Recv"   // DB13
{ S7_Optimized_Access := 'FALSE' }
VERSION : 0.1
   VAR
      Ready : Bool;   // Batch đã sẵn sàng
      Running : Bool;   // Batch đang chạy
      Clock : Bool;   // xung trả về từ cảm biến lưu lượng
      Pulse : Int := 13;   // tổng số xung từ lúc bắt đầu chạy của cảm biến lưu lượng
      Vout : Real;   // thể tích đã xuất ra (m3)
      ctrvalue : Real;   // độ mở van (0-100%)
   END_VAR
BEGIN
END_DATA_BLOCK

DATA_BLOCK "RON922_Send"   // DB14
{ S7_Optimized_Access := 'FALSE' }
VERSION : 0.1
   VAR
      Start : Bool;   // tín hiệu bắt đầu chạy
      Estop : Bool;   // tín hiệu dừng khẩn cấp
      Enable : Bool;   // tín hiệu cho phép làm việc
      PS : Int := 13;   // số xung/lit của cảm biến lưu lượng
      Setpoint : Real;   // thể tích cần xuất
   END_VAR
BEGIN
END_DATA_BLOCK

DATA_BLOCK "RON95_Common"   // DB19
{ S7_Optimized_Access := 'FALSE' }
VERSION : 0.1
   VAR
      Temp : Real := 25.0;   // nhiệt độ (°C)
      Level : Real := 15.0;   // mức (m)
      InitialLevel : Real := 15.0;   // mức ban đầu (m)
      BaseArea : Real := 10.0;   // diện tích đáy (m2)
      Volume : Real;   // thể tích hiện tại (m3)
      InitialVolume : Real;   // thể tích ban đầu (m3)
      Flow1 : Real := 0.0;   // lưu lượng họng 1 (m3/h)
      Flow2 : Real := 0.0;   // lưu lượng họng 2 (m3/h)
   END_VAR
BEGIN
END_DATA_BLOCK

DATA_BLOCK "RON951_Recv"   // DB20
{ S7_Optimized_Access := 'FALSE' }
VERSION : 0.1
   VAR
      Ready : Bool;   // Batch đã sẵn sàng
      Running : Bool;   // Batch đang chạy
      Clock : Bool;   // xung trả về từ cảm biến lưu lượng
      Pulse : Int := 13;   // tổng số xung từ lúc bắt đầu chạy của cảm biến lưu lượng
      Vout : Real;   // thể tích đã xuất ra (m3)
      ctrvalue : Real;   // độ mở van (0-100%)
   END_VAR
BEGIN
END_DATA_BLOCK

DATA_BLOCK "RON951_Send"   // DB21
{ S7_Optimized_Access := 'FALSE' }
VERSION : 0.1
   VAR
      Start : Bool;   // tín hiệu bắt đầu chạy
      Estop : Bool;   // tín hiệu dừng khẩn cấp
      Enable : Bool;   // tín hiệu cho phép làm việc
      PS : Int := 13;   // số xung/lit của cảm biến lưu lượng
      Setpoint : Real;   // thể tích cần xuất
   END_VAR
BEGIN
END_DATA_BLOCK

DATA_BLOCK "RON952_Recv"   // DB22
{ S7_Optimized_Access := 'FALSE' }
VERSION : 0.1
   VAR
      Ready : Bool;   // Batch đã sẵn sàng
      Running : Bool;   // Batch đang chạy
      Clock : Bool;   // xung trả về từ cảm biến lưu lượng
      Pulse : Int := 13;   // tổng số xung từ lúc bắt đầu chạy của cảm biến lưu lượng
      Vout : Real;   // thể tích đã xuất ra (m3)
      ctrvalue : Real;   // độ mở van (0-100%)
   END_VAR
BEGIN
END_DATA_BLOCK

DATA_BLOCK "RON952_Send"   // DB23
{ S7_Optimized_Access := 'FALSE' }
VERSION : 0.1
   VAR
      Start : Bool;   // tín hiệu bắt đầu chạy
      Estop : Bool;   // tín hiệu dừng khẩn cấp
      Enable : Bool;   // tín hiệu cho phép làm việc
      PS : Int := 13;   // số xung/lit của cảm biến lưu lượng
      Setpoint : Real;   // thể tích cần xuất
   END_VAR
BEGIN
END_DATA_BLOCK

DATA_BLOCK "E51_Send"   // DB28
{ S7_Optimized_Access := 'FALSE' }
VERSION : 0.1
   VAR
      Start : Bool;   // tín hiệu bắt đầu chạy
      Estop : Bool;   // tín hiệu dừng khẩn cấp
      Enable : Bool;   // tín hiệu cho phép làm việc
      PS : Int;   // số xung/lit của cảm biến lưu lượng
      Setpoint : Real;   // thể tích cần xuất
   END_VAR
BEGIN
END_DATA_BLOCK

DATA_BLOCK "E51_Recv"   // DB29
{ S7_Optimized_Access := 'FALSE' }
VERSION : 0.1
   VAR
      Ready : Bool;   // Batch đã sẵn sàng
      Running : Bool;   // Batch đang chạy
      ClockRON92 : Bool;   // xung trả về từ cảm biến lưu lượng
      ClockE100 : Bool;   // xung trả về từ cảm biến lưu lượng
      PulseRON92 : Int := 13;   // tổng số xung từ lúc bắt đầu chạy của cảm biến lưu lượng
      PulseE100 : Int := 13;   // tổng số xung từ lúc bắt đầu chạy của cảm biến lưu lượng
      VoutRON92 : Real;   // thể tích đã xuất ra (m3)
      VoutE100 : Real;   // thể tích đã xuất ra (m3)
      Vout : Real;   // thể tích đã xuất ra E5 (m3)
      ctrvalueRON92 : Real;   // độ mở van (0-100%)
      ctrvalueE100 : Real;   // độ mở van (0-100%)
   END_VAR
BEGIN
END_DATA_BLOCK

DATA_BLOCK "E100_Common"   // DB30
{ S7_Optimized_Access := 'FALSE' }
VERSION : 0.1
   VAR
      Temp : Real := 25.0;   // nhiệt độ (°C)
      Level : Real := 15.0;   // mức (m)
      InitialLevel : Real := 15.0;   // mức ban đầu (m)
      BaseArea : Real := 10.0;   // diện tích đáy (m2)
      Volume : Real;   // thể tích hiện tại (m3)
      InitialVolume : Real;   // thể tích ban đầu (m3)
      Flow1 : Real;   // lưu lượng họng 1 (m3/h)
      Flow2 : Real;   // lưu lượng họng 2 (m3/h)
   END_VAR
BEGIN
END_DATA_BLOCK

DATA_BLOCK "E5_Common"   // DB31
{ S7_Optimized_Access := 'FALSE' }
VERSION : 0.1
   VAR
      FlowRON921 : Real;   // lưu lượng họng 1 RON92 (m3/h)
      FlowE1001 : Real;   // lưu lượng họng 1 E100 (m3/h)
      FlowRON922 : Real;   // lưu lượng họng 2 RON92 (m3/h)
      FlowE1002 : Real;   // lưu lượng họng 2 E100 (m3/h)
   END_VAR
BEGIN
END_DATA_BLOCK

DATA_BLOCK "E52_Recv"   // DB32
{ S7_Optimized_Access := 'FALSE' }
VERSION : 0.1
   VAR
      Ready : Bool;   // Batch đã sẵn sàng
      Running : Bool;   // Batch đang chạy
      ClockRON92 : Bool;   // xung trả về từ cảm biến lưu lượng
      ClockE100 : Bool;   // xung trả về từ cảm biến lưu lượng
      PulseRON92 : Int := 13;   // tổng số xung từ lúc bắt đầu chạy của cảm biến lưu lượng
      PulseE100 : Int := 13;   // tổng số xung từ lúc bắt đầu chạy của cảm biến lưu lượng
      VoutRON92 : Real;   // thể tích đã xuất ra (m3)
      VoutE100 : Real;   // thể tích đã xuất ra (m3)
      Vout : Real;   // thể tích đã xuất ra E5 (m3)
      ctrvalueRON92 : Real;   // độ mở van (0-100%)
      ctrvalueE100 : Real;   // độ mở van (0-100%)
   END_VAR
BEGIN
END_DATA_BLOCK

DATA_BLOCK "E52_Send"   // DB33
{ S7_Optimized_Access := 'FALSE' }
VERSION : 0.1
   VAR
      Start : Bool;   // tín hiệu bắt đầu chạy
      Estop : Bool;   // tín hiệu dừng khẩn cấp
      Enable : Bool;   // tín hiệu cho phép làm việc
      PS : Int;   // số xung/lit của cảm biến lưu lượng
      Setpoint : Real;   // thể tích cần xuất
   END_VAR
BEGIN
END_DATA_BLOCK

FUNCTION "DiezelProcess" : Void   // FC1, LAD
{ S7_Optimized_Access := 'TRUE' }
VERSION : 0.1
BEGIN

REGION Network 1: nhận dữ liệu từ DB của BatchController họng 1
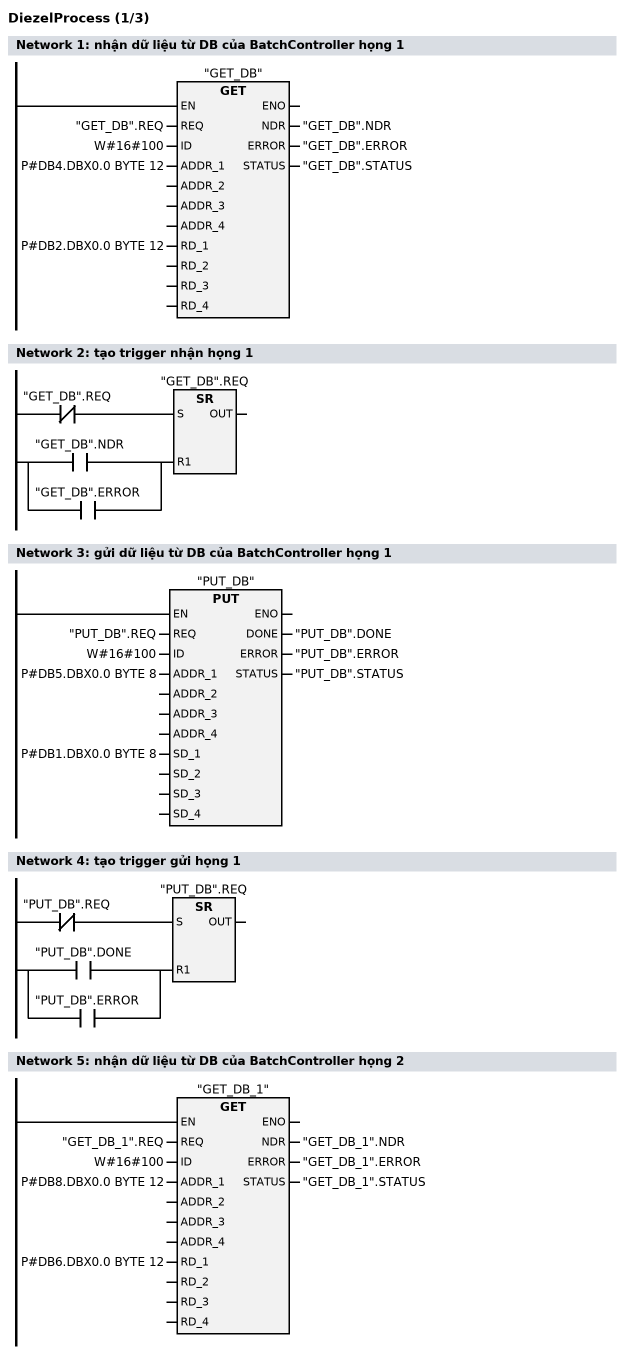
   "GET_DB"(REQ := "GET_DB".REQ,   // GET
            ID := W#16#100,
            ADDR_1 := P#DB4.DBX0.0 BYTE 12,
            RD_1 := P#DB2.DBX0.0 BYTE 12,
            NDR => "GET_DB".NDR,
            ERROR => "GET_DB".ERROR,
            STATUS => "GET_DB".STATUS);
END_REGION

REGION Network 2: tạo trigger nhận họng 1
   RUNG wire#powerrail
      I_Contact( "GET_DB".REQ )
      S_SR(operand := "GET_DB".REQ, r1 := wire#w1)
   END_RUNG
   RUNG wire#powerrail
      Contact( "GET_DB".NDR )
   END_RUNG wire#w1
   RUNG wire#powerrail
      Contact( "GET_DB".ERROR )
   END_RUNG wire#w1
   // the same network as SCL:
   IF NOT "GET_DB".REQ THEN
       "GET_DB".REQ := TRUE;   // SR flip-flop
   END_IF;
   IF "GET_DB".NDR OR "GET_DB".ERROR THEN "GET_DB".REQ := FALSE; END_IF;
END_REGION

REGION Network 3: gửi dữ liệu từ DB của BatchController họng 1
   "PUT_DB"(REQ := "PUT_DB".REQ,   // PUT
            ID := W#16#100,
            ADDR_1 := P#DB5.DBX0.0 BYTE 8,
            SD_1 := P#DB1.DBX0.0 BYTE 8,
            DONE => "PUT_DB".DONE,
            ERROR => "PUT_DB".ERROR,
            STATUS => "PUT_DB".STATUS);
END_REGION

REGION Network 4: tạo trigger gửi họng 1
   RUNG wire#powerrail
      I_Contact( "PUT_DB".REQ )
      S_SR(operand := "PUT_DB".REQ, r1 := wire#w1)
   END_RUNG
   RUNG wire#powerrail
      Contact( "PUT_DB".DONE )
   END_RUNG wire#w1
   RUNG wire#powerrail
      Contact( "PUT_DB".ERROR )
   END_RUNG wire#w1
   // the same network as SCL:
   IF NOT "PUT_DB".REQ THEN
       "PUT_DB".REQ := TRUE;   // SR flip-flop
   END_IF;
   IF "PUT_DB".DONE OR "PUT_DB".ERROR THEN "PUT_DB".REQ := FALSE; END_IF;
END_REGION

REGION Network 5: nhận dữ liệu từ DB của BatchController họng 2
   "GET_DB_1"(REQ := "GET_DB_1".REQ,   // GET
              ID := W#16#100,
              ADDR_1 := P#DB8.DBX0.0 BYTE 12,
              RD_1 := P#DB6.DBX0.0 BYTE 12,
              NDR => "GET_DB_1".NDR,
              ERROR => "GET_DB_1".ERROR,
              STATUS => "GET_DB_1".STATUS);
END_REGION

REGION Network 6: tạo trigger nhận họng 2
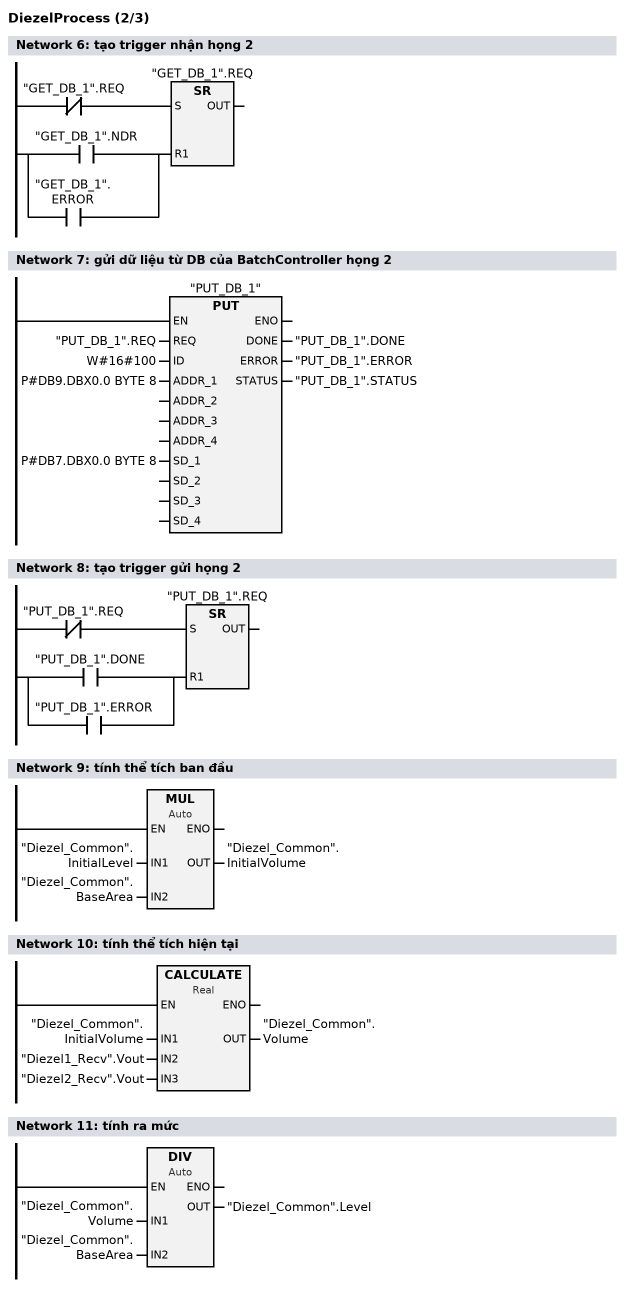
   RUNG wire#powerrail
      I_Contact( "GET_DB_1".REQ )
      S_SR(operand := "GET_DB_1".REQ, r1 := wire#w1)
   END_RUNG
   RUNG wire#powerrail
      Contact( "GET_DB_1".NDR )
   END_RUNG wire#w1
   RUNG wire#powerrail
      Contact( "GET_DB_1".ERROR )
   END_RUNG wire#w1
   // the same network as SCL:
   IF NOT "GET_DB_1".REQ THEN
       "GET_DB_1".REQ := TRUE;   // SR flip-flop
   END_IF;
   IF "GET_DB_1".NDR OR "GET_DB_1".ERROR THEN "GET_DB_1".REQ := FALSE; END_IF;
END_REGION

REGION Network 7: gửi dữ liệu từ DB của BatchController họng 2
   "PUT_DB_1"(REQ := "PUT_DB_1".REQ,   // PUT
              ID := W#16#100,
              ADDR_1 := P#DB9.DBX0.0 BYTE 8,
              SD_1 := P#DB7.DBX0.0 BYTE 8,
              DONE => "PUT_DB_1".DONE,
              ERROR => "PUT_DB_1".ERROR,
              STATUS => "PUT_DB_1".STATUS);
END_REGION

REGION Network 8: tạo trigger gửi họng 2
   RUNG wire#powerrail
      I_Contact( "PUT_DB_1".REQ )
      S_SR(operand := "PUT_DB_1".REQ, r1 := wire#w1)
   END_RUNG
   RUNG wire#powerrail
      Contact( "PUT_DB_1".DONE )
   END_RUNG wire#w1
   RUNG wire#powerrail
      Contact( "PUT_DB_1".ERROR )
   END_RUNG wire#w1
   // the same network as SCL:
   IF NOT "PUT_DB_1".REQ THEN
       "PUT_DB_1".REQ := TRUE;   // SR flip-flop
   END_IF;
   IF "PUT_DB_1".DONE OR "PUT_DB_1".ERROR THEN "PUT_DB_1".REQ := FALSE; END_IF;
END_REGION

REGION Network 9: tính thể tích ban đầu
   RUNG wire#powerrail
      Mul(in1 := "Diezel_Common".InitialLevel, in2 := "Diezel_Common".BaseArea, out => "Diezel_Common".InitialVolume)
   END_RUNG
   // the same network as SCL:
   "Diezel_Common".InitialVolume := "Diezel_Common".InitialLevel * "Diezel_Common".BaseArea;
END_REGION

REGION Network 10: tính thể tích hiện tại
   RUNG wire#powerrail
      { S7_Templates := "SrcType := Real"; S7_Expression := "IN1-IN2-IN3" } Calculate(in1 := "Diezel_Common".InitialVolume, in2 := "Diezel1_Recv".Vout, in3 := "Diezel2_Recv".Vout, out => "Diezel_Common".Volume)
   END_RUNG
   // the same network as SCL:
   "Diezel_Common".Volume := "Diezel_Common".InitialVolume-"Diezel1_Recv".Vout-"Diezel2_Recv".Vout;
END_REGION

REGION Network 11: tính ra mức
   RUNG wire#powerrail
      Div(in1 := "Diezel_Common".Volume, in2 := "Diezel_Common".BaseArea, out => "Diezel_Common".Level)
   END_RUNG
   // the same network as SCL:
   "Diezel_Common".Level := "Diezel_Common".Volume / "Diezel_Common".BaseArea;
END_REGION

REGION Network 12: tính ra lưu lượng họng 1
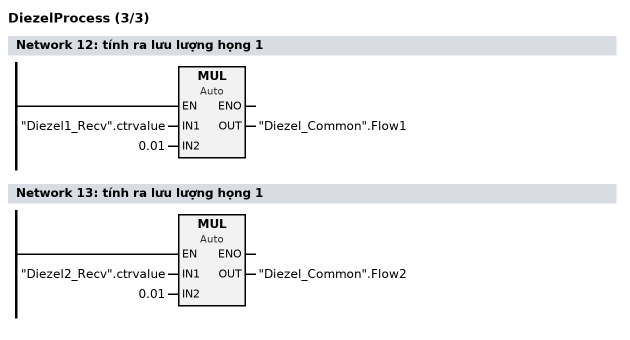
   RUNG wire#powerrail
      Mul(in1 := "Diezel1_Recv".ctrvalue, in2 := 0.01, out => "Diezel_Common".Flow1)
   END_RUNG
   // the same network as SCL:
   "Diezel_Common".Flow1 := "Diezel1_Recv".ctrvalue * 0.01;
END_REGION

REGION Network 13: tính ra lưu lượng họng 1
   RUNG wire#powerrail
      Mul(in1 := "Diezel2_Recv".ctrvalue, in2 := 0.01, out => "Diezel_Common".Flow2)
   END_RUNG
   // the same network as SCL:
   "Diezel_Common".Flow2 := "Diezel2_Recv".ctrvalue * 0.01;
END_REGION
END_FUNCTION

FUNCTION "RON92Process" : Void   // FC2, LAD
{ S7_Optimized_Access := 'TRUE' }
VERSION : 0.1
BEGIN

REGION Network 1: nhận dữ liệu từ DB của BatchController họng 1
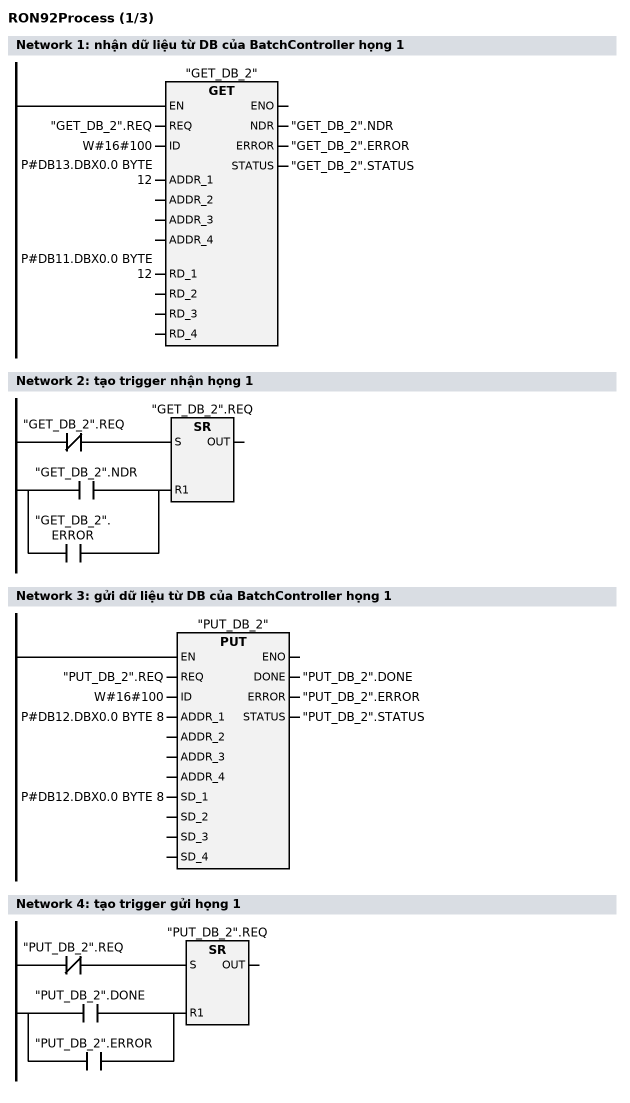
   "GET_DB_2"(REQ := "GET_DB_2".REQ,   // GET
              ID := W#16#100,
              ADDR_1 := P#DB13.DBX0.0 BYTE 12,
              RD_1 := P#DB11.DBX0.0 BYTE 12,
              NDR => "GET_DB_2".NDR,
              ERROR => "GET_DB_2".ERROR,
              STATUS => "GET_DB_2".STATUS);
END_REGION

REGION Network 2: tạo trigger nhận họng 1
   RUNG wire#powerrail
      I_Contact( "GET_DB_2".REQ )
      S_SR(operand := "GET_DB_2".REQ, r1 := wire#w1)
   END_RUNG
   RUNG wire#powerrail
      Contact( "GET_DB_2".NDR )
   END_RUNG wire#w1
   RUNG wire#powerrail
      Contact( "GET_DB_2".ERROR )
   END_RUNG wire#w1
   // the same network as SCL:
   IF NOT "GET_DB_2".REQ THEN
       "GET_DB_2".REQ := TRUE;   // SR flip-flop
   END_IF;
   IF "GET_DB_2".NDR OR "GET_DB_2".ERROR THEN "GET_DB_2".REQ := FALSE; END_IF;
END_REGION

REGION Network 3: gửi dữ liệu từ DB của BatchController họng 1
   "PUT_DB_2"(REQ := "PUT_DB_2".REQ,   // PUT
              ID := W#16#100,
              ADDR_1 := P#DB12.DBX0.0 BYTE 8,
              SD_1 := P#DB12.DBX0.0 BYTE 8,
              DONE => "PUT_DB_2".DONE,
              ERROR => "PUT_DB_2".ERROR,
              STATUS => "PUT_DB_2".STATUS);
END_REGION

REGION Network 4: tạo trigger gửi họng 1
   RUNG wire#powerrail
      I_Contact( "PUT_DB_2".REQ )
      S_SR(operand := "PUT_DB_2".REQ, r1 := wire#w1)
   END_RUNG
   RUNG wire#powerrail
      Contact( "PUT_DB_2".DONE )
   END_RUNG wire#w1
   RUNG wire#powerrail
      Contact( "PUT_DB_2".ERROR )
   END_RUNG wire#w1
   // the same network as SCL:
   IF NOT "PUT_DB_2".REQ THEN
       "PUT_DB_2".REQ := TRUE;   // SR flip-flop
   END_IF;
   IF "PUT_DB_2".DONE OR "PUT_DB_2".ERROR THEN "PUT_DB_2".REQ := FALSE; END_IF;
END_REGION

REGION Network 5: nhận dữ liệu từ DB của BatchController họng 2
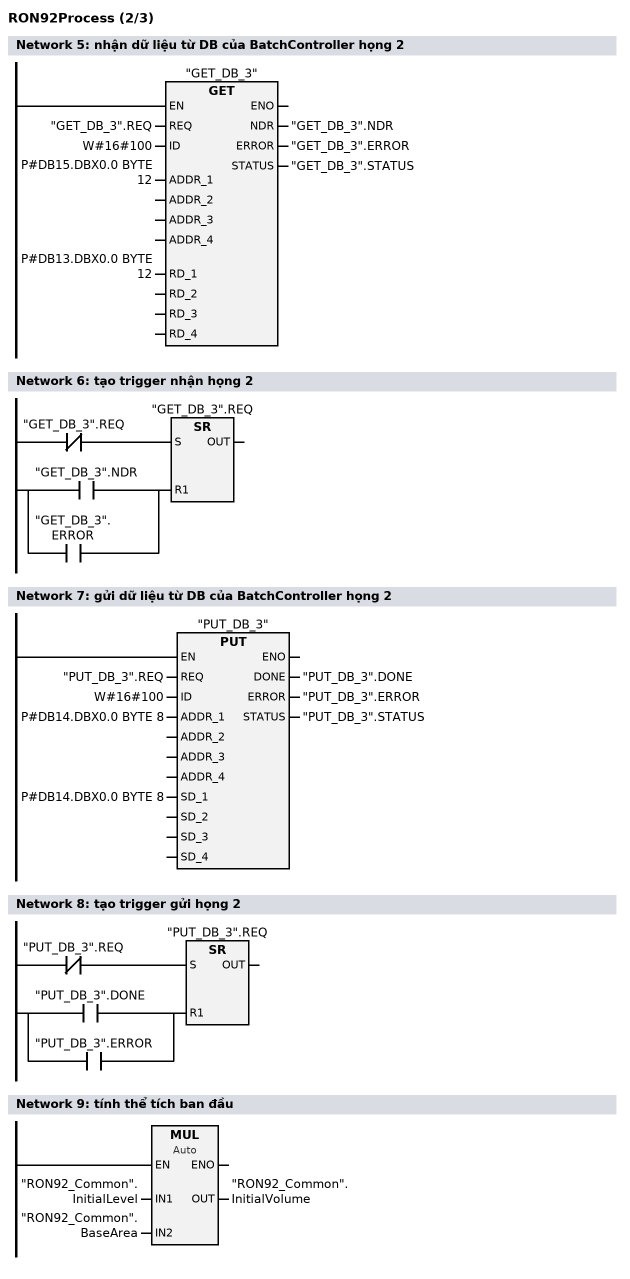
   "GET_DB_3"(REQ := "GET_DB_3".REQ,   // GET
              ID := W#16#100,
              ADDR_1 := P#DB15.DBX0.0 BYTE 12,
              RD_1 := P#DB13.DBX0.0 BYTE 12,
              NDR => "GET_DB_3".NDR,
              ERROR => "GET_DB_3".ERROR,
              STATUS => "GET_DB_3".STATUS);
END_REGION

REGION Network 6: tạo trigger nhận họng 2
   RUNG wire#powerrail
      I_Contact( "GET_DB_3".REQ )
      S_SR(operand := "GET_DB_3".REQ, r1 := wire#w1)
   END_RUNG
   RUNG wire#powerrail
      Contact( "GET_DB_3".NDR )
   END_RUNG wire#w1
   RUNG wire#powerrail
      Contact( "GET_DB_3".ERROR )
   END_RUNG wire#w1
   // the same network as SCL:
   IF NOT "GET_DB_3".REQ THEN
       "GET_DB_3".REQ := TRUE;   // SR flip-flop
   END_IF;
   IF "GET_DB_3".NDR OR "GET_DB_3".ERROR THEN "GET_DB_3".REQ := FALSE; END_IF;
END_REGION

REGION Network 7: gửi dữ liệu từ DB của BatchController họng 2
   "PUT_DB_3"(REQ := "PUT_DB_3".REQ,   // PUT
              ID := W#16#100,
              ADDR_1 := P#DB14.DBX0.0 BYTE 8,
              SD_1 := P#DB14.DBX0.0 BYTE 8,
              DONE => "PUT_DB_3".DONE,
              ERROR => "PUT_DB_3".ERROR,
              STATUS => "PUT_DB_3".STATUS);
END_REGION

REGION Network 8: tạo trigger gửi họng 2
   RUNG wire#powerrail
      I_Contact( "PUT_DB_3".REQ )
      S_SR(operand := "PUT_DB_3".REQ, r1 := wire#w1)
   END_RUNG
   RUNG wire#powerrail
      Contact( "PUT_DB_3".DONE )
   END_RUNG wire#w1
   RUNG wire#powerrail
      Contact( "PUT_DB_3".ERROR )
   END_RUNG wire#w1
   // the same network as SCL:
   IF NOT "PUT_DB_3".REQ THEN
       "PUT_DB_3".REQ := TRUE;   // SR flip-flop
   END_IF;
   IF "PUT_DB_3".DONE OR "PUT_DB_3".ERROR THEN "PUT_DB_3".REQ := FALSE; END_IF;
END_REGION

REGION Network 9: tính thể tích ban đầu
   RUNG wire#powerrail
      Mul(in1 := "RON92_Common".InitialLevel, in2 := "RON92_Common".BaseArea, out => "RON92_Common".InitialVolume)
   END_RUNG
   // the same network as SCL:
   "RON92_Common".InitialVolume := "RON92_Common".InitialLevel * "RON92_Common".BaseArea;
END_REGION

REGION Network 10: tính thể tích hiện tại
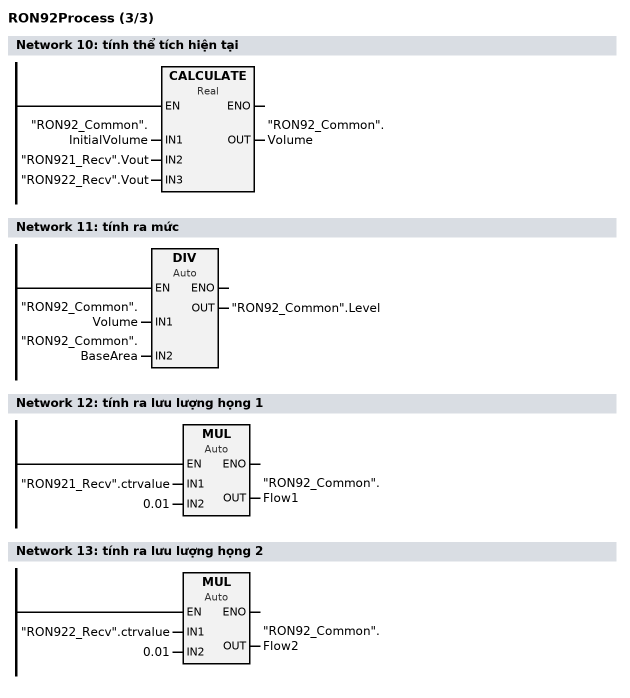
   RUNG wire#powerrail
      { S7_Templates := "SrcType := Real"; S7_Expression := "IN1-IN2-IN3" } Calculate(in1 := "RON92_Common".InitialVolume, in2 := "RON921_Recv".Vout, in3 := "RON922_Recv".Vout, out => "RON92_Common".Volume)
   END_RUNG
   // the same network as SCL:
   "RON92_Common".Volume := "RON92_Common".InitialVolume-"RON921_Recv".Vout-"RON922_Recv".Vout;
END_REGION

REGION Network 11: tính ra mức
   RUNG wire#powerrail
      Div(in1 := "RON92_Common".Volume, in2 := "RON92_Common".BaseArea, out => "RON92_Common".Level)
   END_RUNG
   // the same network as SCL:
   "RON92_Common".Level := "RON92_Common".Volume / "RON92_Common".BaseArea;
END_REGION

REGION Network 12: tính ra lưu lượng họng 1
   RUNG wire#powerrail
      Mul(in1 := "RON921_Recv".ctrvalue, in2 := 0.01, out => "RON92_Common".Flow1)
   END_RUNG
   // the same network as SCL:
   "RON92_Common".Flow1 := "RON921_Recv".ctrvalue * 0.01;
END_REGION

REGION Network 13: tính ra lưu lượng họng 2
   RUNG wire#powerrail
      Mul(in1 := "RON922_Recv".ctrvalue, in2 := 0.01, out => "RON92_Common".Flow2)
   END_RUNG
   // the same network as SCL:
   "RON92_Common".Flow2 := "RON922_Recv".ctrvalue * 0.01;
END_REGION
END_FUNCTION

FUNCTION "RON95Process" : Void   // FC3, LAD
{ S7_Optimized_Access := 'TRUE' }
VERSION : 0.1
BEGIN

REGION Network 1: nhận dữ liệu từ DB của BatchController họng 1
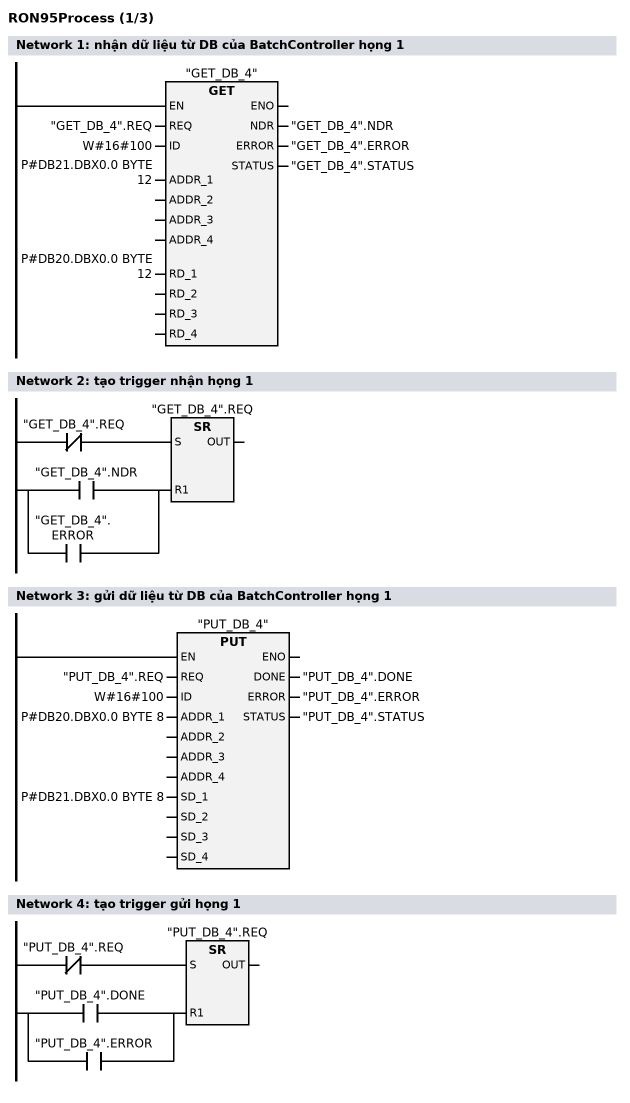
   "GET_DB_4"(REQ := "GET_DB_4".REQ,   // GET
              ID := W#16#100,
              ADDR_1 := P#DB21.DBX0.0 BYTE 12,
              RD_1 := P#DB20.DBX0.0 BYTE 12,
              NDR => "GET_DB_4".NDR,
              ERROR => "GET_DB_4".ERROR,
              STATUS => "GET_DB_4".STATUS);
END_REGION

REGION Network 2: tạo trigger nhận họng 1
   RUNG wire#powerrail
      I_Contact( "GET_DB_4".REQ )
      S_SR(operand := "GET_DB_4".REQ, r1 := wire#w1)
   END_RUNG
   RUNG wire#powerrail
      Contact( "GET_DB_4".NDR )
   END_RUNG wire#w1
   RUNG wire#powerrail
      Contact( "GET_DB_4".ERROR )
   END_RUNG wire#w1
   // the same network as SCL:
   IF NOT "GET_DB_4".REQ THEN
       "GET_DB_4".REQ := TRUE;   // SR flip-flop
   END_IF;
   IF "GET_DB_4".NDR OR "GET_DB_4".ERROR THEN "GET_DB_4".REQ := FALSE; END_IF;
END_REGION

REGION Network 3: gửi dữ liệu từ DB của BatchController họng 1
   "PUT_DB_4"(REQ := "PUT_DB_4".REQ,   // PUT
              ID := W#16#100,
              ADDR_1 := P#DB20.DBX0.0 BYTE 8,
              SD_1 := P#DB21.DBX0.0 BYTE 8,
              DONE => "PUT_DB_4".DONE,
              ERROR => "PUT_DB_4".ERROR,
              STATUS => "PUT_DB_4".STATUS);
END_REGION

REGION Network 4: tạo trigger gửi họng 1
   RUNG wire#powerrail
      I_Contact( "PUT_DB_4".REQ )
      S_SR(operand := "PUT_DB_4".REQ, r1 := wire#w1)
   END_RUNG
   RUNG wire#powerrail
      Contact( "PUT_DB_4".DONE )
   END_RUNG wire#w1
   RUNG wire#powerrail
      Contact( "PUT_DB_4".ERROR )
   END_RUNG wire#w1
   // the same network as SCL:
   IF NOT "PUT_DB_4".REQ THEN
       "PUT_DB_4".REQ := TRUE;   // SR flip-flop
   END_IF;
   IF "PUT_DB_4".DONE OR "PUT_DB_4".ERROR THEN "PUT_DB_4".REQ := FALSE; END_IF;
END_REGION

REGION Network 5: nhận dữ liệu từ DB của BatchController họng 2
